// TIA Portal project "ELEVEYTOR" (V15.1)

(* hardware
DEVICE "S7-1200 station_1"  S7-1200 Station
   slot 0: "Rack_0"  S7-1200 Rack  Rack  V1.0
   slot 1: "PLC_1"  CPU 1214C AC/DC/Rly  6ES7 214-1BG40-0XB0  V4.2
   slot 2: "DI 16/DQ 16x24VDC_1"  6ES7 223-1BL32-0XB0  V2.0
DEVICE "PC-System_1"  SIMATIC PC station
   slot 0: "SIMATIC PC station"  Rail  SIMATIC PC-Station  V1.0
      slot 125: "Stationmanager"  Station_Manager  V6.0.4
   slot 1: "HMI_RT_1"  WinCC RT Advanced  6AV2 104-0xxxx-xxxx  15.1.0.0
      slot 33792: "Host interface"  Host interface
   slot 2: "IE general_1"  IE General  IE_CP  V8.2.0
*)

// ===== PLC "PLC_1"  CPU 1214C AC/DC/Rly =====

VAR_GLOBAL   // PLC tag table "Default tag table"
   "System_Byte" AT %MB1 : Byte;
   "FirstScan" AT %M1.0 : Bool;
   "DiagStatusUpdate" AT %M1.1 : Bool;
   "AlwaysTRUE" AT %M1.2 : Bool;
   "AlwaysFALSE" AT %M1.3 : Bool;
   "Clock_Byte" AT %MB0 : Byte;
   "Clock_10Hz" AT %M0.0 : Bool;
   "Clock_5Hz" AT %M0.1 : Bool;
   "Clock_2.5Hz" AT %M0.2 : Bool;
   "Clock_2Hz" AT %M0.3 : Bool;
   "Clock_1.25Hz" AT %M0.4 : Bool;
   "Clock_1Hz" AT %M0.5 : Bool;
   "Clock_0.625Hz" AT %M0.6 : Bool;
   "Clock_0.5Hz" AT %M0.7 : Bool;
   "Tag_1" AT %M900.0 : Bool;
   "Led" AT %MB6 : Byte;
END_VAR

VAR_GLOBAL   // PLC tag table "PRIORITIZE"
   "PRIORITIZE_1" AT %MB50 : SInt;   // Gọi lên x1, gọi xuống x0 (21,31, 41,51...20,30,40,50)
   "PRIORITIZE_2" AT %MB51 : SInt;
   "PRIORITIZE_3" AT %MB52 : SInt;
   "PRIORITIZE_4" AT %MB53 : SInt;
   "PRIORITIZE_5" AT %MB54 : SInt;
   "PRIORITIZE_6" AT %MB55 : SInt;
   "PRIORITIZE_SHIFT_1" AT %MD50 : DInt;
   "PRIORITIZE_SHIFT_2" AT %MD53 : DInt;
   "PRIORITIZE_SHIFT_3" AT %MD56 : DInt;
   "PRIORITIZE_7" AT %MB56 : SInt;
   "PRIORITIZE_8" AT %MB57 : SInt;
   "PRIORITIZE_9" AT %MB58 : SInt;
   "PRIORITIZE_10" AT %MB59 : SInt;
   "PRIORITIZE_11" AT %MB60 : SInt;
   "PRIORITIZE_12" AT %MB61 : SInt;
   "PRIORITIZE_SHIFT_4" AT %MD59 : DInt;
   "PRIORITIZE_POSITION" AT %MW70 : Int;
   "PRIORITIZE_13_Addition" AT %MB63 : SInt;   // Khi một tầng chọn cả lên và xuống thì dùng
   "PRIORITIZE_14_Addition" AT %MB64 : SInt;   // Spare
   "PRIORITIZE_15_Addition" AT %MB65 : SInt;   // Spare
   "PRIORITIZE_16_Addition" AT %MB66 : SInt;   // Spare
   "PRIORITIZE_SHIFT_5" AT %MD62 : DInt;
END_VAR

VAR_GLOBAL   // PLC tag table "OUTPUT"
   "Q_Lamp_System" AT %Q0.0 : Bool;   // Đèn làm việc
   "Q_Cabinet_Up" AT %Q0.1 : Bool;   // Buồng thang đi lên
   "Q_Cabinet_Down" AT %Q0.2 : Bool;   // Buồng thang đi xuống
   "Q_Door_Open" AT %Q0.3 : Bool;   // Cửa buồng thang mở
   "Q_Door_Close" AT %Q0.4 : Bool;   // Cửa buồng thang đóng
   "Q_BTT_Up_F1" AT %Q0.5 : Bool;   // Đèn nút nhấn đi lên F1
   "Q_BTT_Up_F2" AT %Q0.6 : Bool;   // Đèn nút nhấn đi lên F2
   "Q_BTT_Up_F3" AT %Q0.7 : Bool;   // Đèn nút nhấn đi lên F3
   "Q_BTT_Up_F4" AT %Q1.0 : Bool;   // Đèn nút nhấn đi lên F4
   "Q_BTT_Up_F5" AT %Q1.1 : Bool;   // Đèn nút nhấn đi lên F5
   "Q_BTT_Down_F2" AT %Q1.2 : Bool;   // Đèn nút nhấn đi xuống F2
   "Q_BTT_Down_F3" AT %Q1.3 : Bool;   // Đèn nút nhấn đi xuống F3
   "Q_BTT_Down_F4" AT %Q1.4 : Bool;   // Đèn nút nhấn đi xuống F4
   "Q_BTT_Down_F5" AT %Q1.5 : Bool;   // Đèn nút nhấn đi xuống F5
   "Q_BTT_Down_F6" AT %Q1.6 : Bool;   // Đèn nút nhấn đi xuống F6
   "Q_BTT_CABIN_F1" AT %Q1.7 : Bool;   // Đèn nút nhấn trong buồng thang F1
   "Q_BTT_CABIN_F2" AT %Q2.0 : Bool;   // Đèn nút nhấn trong buồng thang F2
   "Q_BTT_CABIN_F3" AT %Q2.1 : Bool;   // Đèn nút nhấn trong buồng thang F3
   "Q_BTT_CABIN_F4" AT %Q2.2 : Bool;   // Đèn nút nhấn trong buồng thang F4
   "Q_BTT_CABIN_F5" AT %Q2.3 : Bool;   // Đèn nút nhấn trong buồng thang F5
   "Q_BTT_CABIN_F6" AT %Q2.4 : Bool;   // Đèn nút nhấn trong buồng thang F6
   "Q_Lamp_Weight_Alarm" AT %Q2.5 : Bool;   // Đèn cảnh báo quá trọng lượng
END_VAR

VAR_GLOBAL   // PLC tag table "INPUT"
   "I_BTT_DOOR_OPEN" AT %I1.4 : Bool;   // Nút nhấn mở cửa
   "I_BTT_DOOR_CLOSE" AT %I2.7 : Bool;   // Nút nhấn đóng cửa
   "I_BTT_CABINET_F1" AT %I0.5 : Bool;   // Nút nhấn chọn tầng trong thang máy Tầng 1
   "I_BTT_CABINET_F2" AT %I0.3 : Bool;   // Nút nhấn chọn tầng trong thang máy Tầng 2
   "I_BTT_CABINET_F3" AT %I0.2 : Bool;   // Nút nhấn chọn tầng trong thang máy Tầng 3
   "I_BTT_CABINET_F4" AT %I0.4 : Bool;   // Nút nhấn chọn tầng trong thang máy Tầng 4
   "I_BTT_UP_F1" AT %I1.2 : Bool;   // Nút nhấn đi lên/xuống tầng 1
   "I_BTT_UP_F2" AT %I0.6 : Bool;   // Nút nhấn đi lên tầng 2
   "I_BTT_UP_F3" AT %I1.0 : Bool;   // Nút nhấn đi lên tầng 3
   "I_BTT_DOWN_F2" AT %I1.3 : Bool;   // Nút nhấn đi xuống tầng 2
   "I_BTT_DOWN_F3" AT %I0.7 : Bool;   // Nút nhấn đi xuống tầng 3
   "I_BTT_DOWN_F4" AT %I1.1 : Bool;   // Nút nhấn đi xuống tầng 4
   "I_LS_DOOR_OPENED" AT %I2.5 : Bool;   // Công tắc hành trình mở cửa
   "I_LS_DOOR_CLOSED" AT %I2.4 : Bool;   // Công tắc hành trình đóng cửa
   "I_BTT_MAN_CABINET_UP" AT %I3.0 : Bool;   // Nút nhấn cabinet nâng chế độ bằng tay
   "I_BTT_MAN_CABINET_DOWN" AT %I2.6 : Bool;   // Nút nhấn cabinet hạ chế độ bằng tay
   "I_BTT_MAN_DOOR_OPEN" AT %I3.1 : Bool;   // Nút nhấn mở cửa chế độ bằng tay
   "I_BTT_MAN_DOOR_CLOSE" AT %I3.5 : Bool;   // nút nhấn đóng cửa chế độ bằng tay
   "I_SW_AUTO" AT %I3.6 : Bool;   // Switch chọn chế độ tự động
   "I_SW_MANU" AT %I3.2 : Bool;   // Switch chọn chế độ bằng tay
   "ID0" AT %ID0 : DWord;
   "I_BTT_MAN_CABIN_STOP" AT %I13.3 : Bool;
   "I_LS_CABINET_2" AT %I2.1 : Bool;
   "I_LS_CABINET_3" AT %I2.2 : Bool;
   "I_LS_CABINET_4" AT %I2.3 : Bool;
   "I_LS_CABINET_1" AT %I2.0 : Bool;
END_VAR

VAR_GLOBAL   // PLC tag table "MEMORY"
   "M_BTT_DOOR_OPEN" AT %M10.0 : Bool;
   "M_BTT_DOOR_CLOSE" AT %M10.1 : Bool;
   "M_BTT_CABINET_F1" AT %M10.2 : Bool;
   "M_BTT_CABINET_F2" AT %M10.3 : Bool;
   "M_BTT_CABINET_F3" AT %M10.4 : Bool;
   "M_BTT_CABINET_F4" AT %M10.5 : Bool;
   "M_BTT_CABINET_F5" AT %M10.6 : Bool;
   "M_BTT_CABINET_F6" AT %M10.7 : Bool;
   "M_BTT_UP_F1" AT %M11.0 : Bool;
   "M_BTT_UP_F2" AT %M11.1 : Bool;
   "M_BTT_UP_F3" AT %M11.2 : Bool;
   "M_BTT_UP_F4" AT %M11.3 : Bool;
   "M_BTT_UP_F5" AT %M11.4 : Bool;
   "M_BTT_DOWN_F2" AT %M11.5 : Bool;
   "M_BTT_DOWN_F3" AT %M11.6 : Bool;
   "M_BTT_DOWN_F4" AT %M11.7 : Bool;
   "M_BTT_DOWN_F5" AT %M12.0 : Bool;
   "M_BTT_DOWN_F6" AT %M12.1 : Bool;
   "M_LS_CABINET" AT %M12.2 : Bool;
   "M_LS_DOOR_OPENED" AT %M12.3 : Bool;
   "M_LS_DOOR_CLOSED" AT %M12.4 : Bool;
   "M_BTT_MAN_CABINET_UP" AT %M12.5 : Bool;
   "M_BTT_MAN_CABINET_DOWN" AT %M12.6 : Bool;
   "M_BTT_MAN_DOOR_OPEN" AT %M12.7 : Bool;
   "M_BTT_MAN_DOOR_CLOSE" AT %M13.0 : Bool;
   "M_SW_AUTO" AT %M13.1 : Bool;
   "M_SW_MANU" AT %M13.2 : Bool;
   "M_BTT_Simulation" AT %M300.0 : Bool;
   "MD10" AT %MD10 : DWord;
   "M_BTT_MAN_DOOR_STOP" AT %M13.4 : Bool;
   "M_BTT_MAN_CABIN_STOP" AT %M13.3 : Bool;
END_VAR

DATA_BLOCK "DB_Status"   // DB1
{ S7_Optimized_Access := 'FALSE' }
VERSION : 0.1
   VAR
      PRIOTIZE_1 : SInt;
      PRIOTIZE_2 : SInt;
      PRIOTIZE_3 : SInt;
      PRIOTIZE_4 : SInt;
      PRIOTIZE_5 : SInt;
      PRIOTIZE_6 : SInt;
      PRIOTIZE_7 : SInt;
      PRIOTIZE_8 : SInt;
      PRIOTIZE_9 : SInt;
      PRIOTIZE_10 : SInt;
      PRIOTIZE_11 : SInt;
      PRIOTIZE_12 : SInt;
      PRIOTIZE_13 : SInt;
      PRIOTIZE_14 : SInt;
      PRIOTIZE_15 : SInt;
      PRIOTIZE_16 : SInt;
      PRIOTIZE_17 : SInt;
      PRIOTIZE_18 : SInt;
      PRIOTIZE_19 : SInt;
      PRIOTIZE_20 : SInt;
      LS_F1 : Bool;
      LS_F2 : Bool;
      LS_F3 : Bool;
      LS_F4 : Bool;
      LS_F5 : Bool;
      LS_F6 : Bool;
      LS_F7 : Bool;   // Spare
      LS_F8 : Bool;   // Spare
      LS_F9 : Bool;   // Spare
      LS_F10 : Bool;   // Spare
      Up_Called_F1 : Bool;
      Up_Called_F2 : Bool;
      Up_Called_F3 : Bool;
      Up_Called_F4 : Bool;
      Up_Called_F5 : Bool;
      Up_Called_F6 : Bool;
      Down_Called_F1 : Bool;
      Down_Called_F2 : Bool;
      Down_Called_F3 : Bool;
      Down_Called_F4 : Bool;
      Down_Called_F5 : Bool;
      Down_Called_F6 : Bool;
      Q_Lamp_System : Bool;
      Q_Cabinet_Up : Bool;
      Q_Cabinet_Down : Bool;
      Q_Door_Open : Bool;
      Q_Door_Close : Bool;
      Q_BTT_Up_F1 : Bool;
      Q_BTT_Up_F2 : Bool;
      Q_BTT_Up_F3 : Bool;
      Q_BTT_Up_F4 : Bool;
      Q_BTT_Up_F5 : Bool;
      Q_BTT_Down_F2 : Bool;
      Q_BTT_Down_F3 : Bool;
      Q_BTT_Down_F4 : Bool;
      Q_BTT_Down_F5 : Bool;
      Q_BTT_Down_F6 : Bool;
      DOOR_Delay_Open : Bool;
      CABINET_AT_FLOOR : Int;
      Actual_Weight : Real;
      CABIN_LastStatus_Upping : Bool;   // Trước đó buồng thang đi lên (trạng thái)
      CABIN_LastStatus_Dowing : Bool;   // Trước đó buồng thang đi xuống (trạng thái)
   END_VAR
BEGIN
END_DATA_BLOCK

DATA_BLOCK "DB_PRIOTIZE"   // DB2
{ S7_Optimized_Access := 'TRUE' }
VERSION : 0.1
BEGIN
END_DATA_BLOCK

DATA_BLOCK "DB_Command"   // DB3
{ S7_Optimized_Access := 'TRUE' }
VERSION : 0.1
   VAR
      F1_Up_Seleced : Bool;
      F2_Up_Seleced : Bool;
      F3_Up_Seleced : Bool;
      F4_Up_Seleced : Bool;
      F5_Up_Seleced : Bool;
      F2_Down_Seleced : Bool;
      F3_Down_Seleced : Bool;
      F4_Down_Seleced : Bool;
      F5_Down_Seleced : Bool;
      F6_Down_Seleced : Bool;
      F1_Selected : Bool;
      F2_Selected : Bool;
      F3_Selected : Bool;
      F4_Selected : Bool;
      F5_Selected : Bool;
      F6_Selected : Bool;
      F_Rq_Cabin_Stop : Bool;   // Yêu cầu dừng cabin FC tầng gọi cuối cùng
      F_Rq_Door_Open : Bool;   // Yêu cầu mở cửa FC tầng gọi cuối cùng
      F_Rq_Clear_Priotize : Bool;   // Yêu cầu xóa ưu tiên FC tầng gọi cuối cùng
   END_VAR
BEGIN
END_DATA_BLOCK

DATA_BLOCK "PULSE"   // DB4
{ S7_Optimized_Access := 'TRUE' }
VERSION : 0.1
   VAR
      FC2_F1_P1 : Bool;
      FC2_F1_P2 : Bool;
      FC2_F2_P1 : Bool;
      FC2_F2_P2 : Bool;
      FC2_F3_P1 : Bool;
      FC2_F3_P2 : Bool;
      FC2_F4_P1 : Bool;
      FC2_F4_P2 : Bool;
      FC2_F5_P1 : Bool;
      FC2_F5_P2 : Bool;
      FC2_F6_P1 : Bool;
      FC2_F6_P2 : Bool;
      FC1_P1 : Bool;
      FC1_P2 : Bool;
      F1_Upping_P1 : Bool;
      F1_Upping_P2 : Bool;
      F2_Upping_P1 : Bool;
      F2_Upping_P2 : Bool;
      F3_Upping_P1 : Bool;
      F3_Upping_P2 : Bool;
      F4_Upping_P1 : Bool;
      F4_Upping_P2 : Bool;
      F5_Upping_P1 : Bool;
      F5_Upping_P2 : Bool;
      F6_Upping_P1 : Bool;
      F6_Upping_P2 : Bool;
      F1_Downing_P1 : Bool;
      F1_Downing_P2 : Bool;
      F2_Downing_P1 : Bool;
      F2_Downing_P2 : Bool;
      F3_Downing_P1 : Bool;
      F3_Downing_P2 : Bool;
      F4_Downing_P1 : Bool;
      F4_Downing_P2 : Bool;
      F5_Downing_P1 : Bool;
      F5_Downing_P2 : Bool;
      F6_Downing_P1 : Bool;
      F6_Downing_P2 : Bool;
      FC7_N1 : Bool;
      FC7_P1 : Bool;
      FC7_P2 : Bool;
      FC7_P3 : Bool;
      FC7_P4 : Bool;
      FC7_N2 : Bool;
      FC7_P5 : Bool;
      FC7_Pulse_Door_Lock : Bool;
      FC7_N3 : Bool;
      FC12_Pulse_2S : Bool;
      "2Second_Pulse_Upping_F1" : Bool;
      "2Second_Pulse_Upping_F2" : Bool;
      "2Second_Pulse_Upping_F3" : Bool;
      "2Second_Pulse_Upping_F4" : Bool;
      "2Second_Pulse_Upping_F5" : Bool;
      "2Second_Pulse_Upping_F6" : Bool;
      "2Second_Pulse_Downing_F1" : Bool;
      "2Second_Pulse_Downing_F2" : Bool;
      "2Second_Pulse_Downing_F3" : Bool;
      "2Second_Pulse_Downing_F4" : Bool;
      "2Second_Pulse_Downing_F5" : Bool;
      "2Second_Pulse_Downing_F6" : Bool;
      FC4_Temp_Pulse : Bool;
      FC12_Pulse_Up_F1 : Bool;
      FC12_Pulse_Up_F2 : Bool;
      FC12_Pulse_Up_F3 : Bool;
      FC12_Pulse_Up_F4 : Bool;
      FC12_Pulse_Up_F5 : Bool;
      FC12_Pulse_Up_F6 : Bool;
      FC12_Pulse_Down_F1 : Bool;
      FC12_Pulse_Down_F2 : Bool;
      FC12_Pulse_Down_F3 : Bool;
      FC12_Pulse_Down_F4 : Bool;
      FC12_Pulse_Down_F5 : Bool;
      FC12_Pulse_Down_F6 : Bool;
      FC7_Pulse_Door_Lock_Temp : Bool;
      FC8_P1 : Bool;
      FC8_P2 : Bool;
      FC1_P3 : Bool;
      FC1_Shift_Request : Bool;
   END_VAR
BEGIN
END_DATA_BLOCK

DATA_BLOCK "DB_FRECONDITION"   // DB5
{ S7_Optimized_Access := 'TRUE' }
VERSION : 0.1
   VAR
      DOOR_Open : Bool;
      DOOR_Permit_time : Bool;
   END_VAR
BEGIN
END_DATA_BLOCK

DATA_BLOCK "DB_SETTING"   // DB6
{ S7_Optimized_Access := 'TRUE' }
VERSION : 0.1
   VAR RETAIN
      Weight : Real := 1000.0;
      Door_Open_Time : Time := T#5ms;
      Extreme_Time : Time := T#5ms;
   END_VAR
BEGIN
END_DATA_BLOCK

DATA_BLOCK "DB_SIMULATION"   // DB8
{ S7_Optimized_Access := 'TRUE' }
VERSION : 0.1
   VAR
      POS_CABINET : Int;
      POS_DOOR : Int;
      DOOR_F1 : Int;   // THANG MÁY Ở TẦNG 1
      DOOR_F2 : Int;   // THANG MÁY Ở TẦNG 2
      DOOR_F3 : Int;   // THANG MÁY Ở TẦNG 3
      DOOR_F4 : Int;   // THANG MÁY Ở TẦNG 4
      Weight : DInt;
   END_VAR
BEGIN
END_DATA_BLOCK

DATA_BLOCK "Display_number_DB"   // DB15
{ S7_Optimized_Access := 'TRUE' }
VERSION : 0.1
// stored: InstanceOfName Display_number
"Display_number"
BEGIN
END_DATA_BLOCK

// folder: System blocks/Program resources

DATA_BLOCK "DELAY_OPEN"   // DB7
{ S7_Optimized_Access := 'TRUE' }
AUTHOR : Simatic
FAMILY : IEC
NAME : IEC_TMR
VERSION : 1.0
// stored: InstanceOfName IEC_TIMER
"IEC_TIMER"
BEGIN
END_DATA_BLOCK

DATA_BLOCK "SIMU_CABINET"   // DB9
{ S7_Optimized_Access := 'TRUE' }
AUTHOR : Simatic
FAMILY : IEC
NAME : CNTR
VERSION : 1.0
// stored: InstanceOfName IEC_COUNTER
"IEC_COUNTER"
BEGIN
END_DATA_BLOCK

DATA_BLOCK "SIMU_DOOR"   // DB10
{ S7_Optimized_Access := 'TRUE' }
AUTHOR : Simatic
FAMILY : IEC
NAME : CNTR
VERSION : 1.0
// stored: InstanceOfName IEC_COUNTER
"IEC_COUNTER"
BEGIN
END_DATA_BLOCK

DATA_BLOCK "DOOR_EXTREME"   // DB11
{ S7_Optimized_Access := 'TRUE' }
AUTHOR : Simatic
FAMILY : IEC
NAME : IEC_TMR
VERSION : 1.0
// stored: InstanceOfName IEC_TIMER
"IEC_TIMER"
BEGIN
END_DATA_BLOCK

DATA_BLOCK "FC12_DELAY_2S"   // DB12
{ S7_Optimized_Access := 'TRUE' }
AUTHOR : Simatic
FAMILY : IEC
NAME : IEC_TMR
VERSION : 1.0
// stored: InstanceOfName IEC_TIMER
"IEC_TIMER"
BEGIN
END_DATA_BLOCK

DATA_BLOCK "FC4_PULSE_2S"   // DB13
{ S7_Optimized_Access := 'TRUE' }
AUTHOR : Simatic
FAMILY : IEC
NAME : IEC_TMR
VERSION : 1.0
// stored: InstanceOfName IEC_TIMER
"IEC_TIMER"
BEGIN
END_DATA_BLOCK

DATA_BLOCK "PULSE_DOOR_LOCK"   // DB14
{ S7_Optimized_Access := 'TRUE' }
AUTHOR : Simatic
FAMILY : IEC
NAME : IEC_TMR
VERSION : 1.0
// stored: InstanceOfName IEC_TIMER
"IEC_TIMER"
BEGIN
END_DATA_BLOCK

// folder: (top level)

FUNCTION_BLOCK "Display_number"   // FB1, SCL
{ S7_Optimized_Access := 'TRUE' }
VERSION : 0.1
   VAR_INPUT
      BCD : Int;
   END_VAR
   VAR_OUTPUT
      LED : Byte;
   END_VAR
   VAR_TEMP
      TMP : Byte;
   END_VAR
BEGIN
   CASE #BCD OF
       1:  // Statement section case 1
           #TMP := 16#6;
       2:  // Statement section case 1
           #TMP := 16#5B;
       3:  // Statement section case 1
           #TMP := 16#4F;
       4:  // Statement section case 1
           #TMP := 16#66;

       ELSE  // Statement section ELSE
           ;
   END_CASE;
   #LED := #TMP;
END_FUNCTION_BLOCK

FUNCTION "1.FC_SHIFT" : Void   // FC1, LAD
{ S7_Optimized_Access := 'TRUE' }
VERSION : 0.1
// 1. Network 1 là lệnh shift word (tức là di chuyển chể độ ưu tiên), ở đây sẽ có 6 chế độ ưu tiên, tầng nào ưu tiên nhất thì sẽ ưu tiên tầng đó.
// Bit shift sẽ thực hiện khi:
// 1.1. Thang máy chạm công tắc hành trình của một tầng nào đó
// 1.2. Cửa buồng thang mở
// >>> tất nhiên với điều kiện ở ô nhớ ưu tiên 1 không phải là tầng đó, ví dụ đang ở tầng 2 mà ô nhớ ưu tiên 1 có giá trị là 2 thì mới shift, còn không thì thôi.
// 
// >>> Nếu giá trị ưu tiên đầu tiên mà bằng 0 thì tiến hành shift các miền nhớ khác tiến về trước mỗi 100ms (Clock_10Hz)
   VAR_TEMP   // added for the SCL form of the ladder/FBD networks
      _w1 : Bool;
      _w2 : Bool;
   END_VAR
BEGIN

REGION Network 1: SHIFT PRIORITIZE
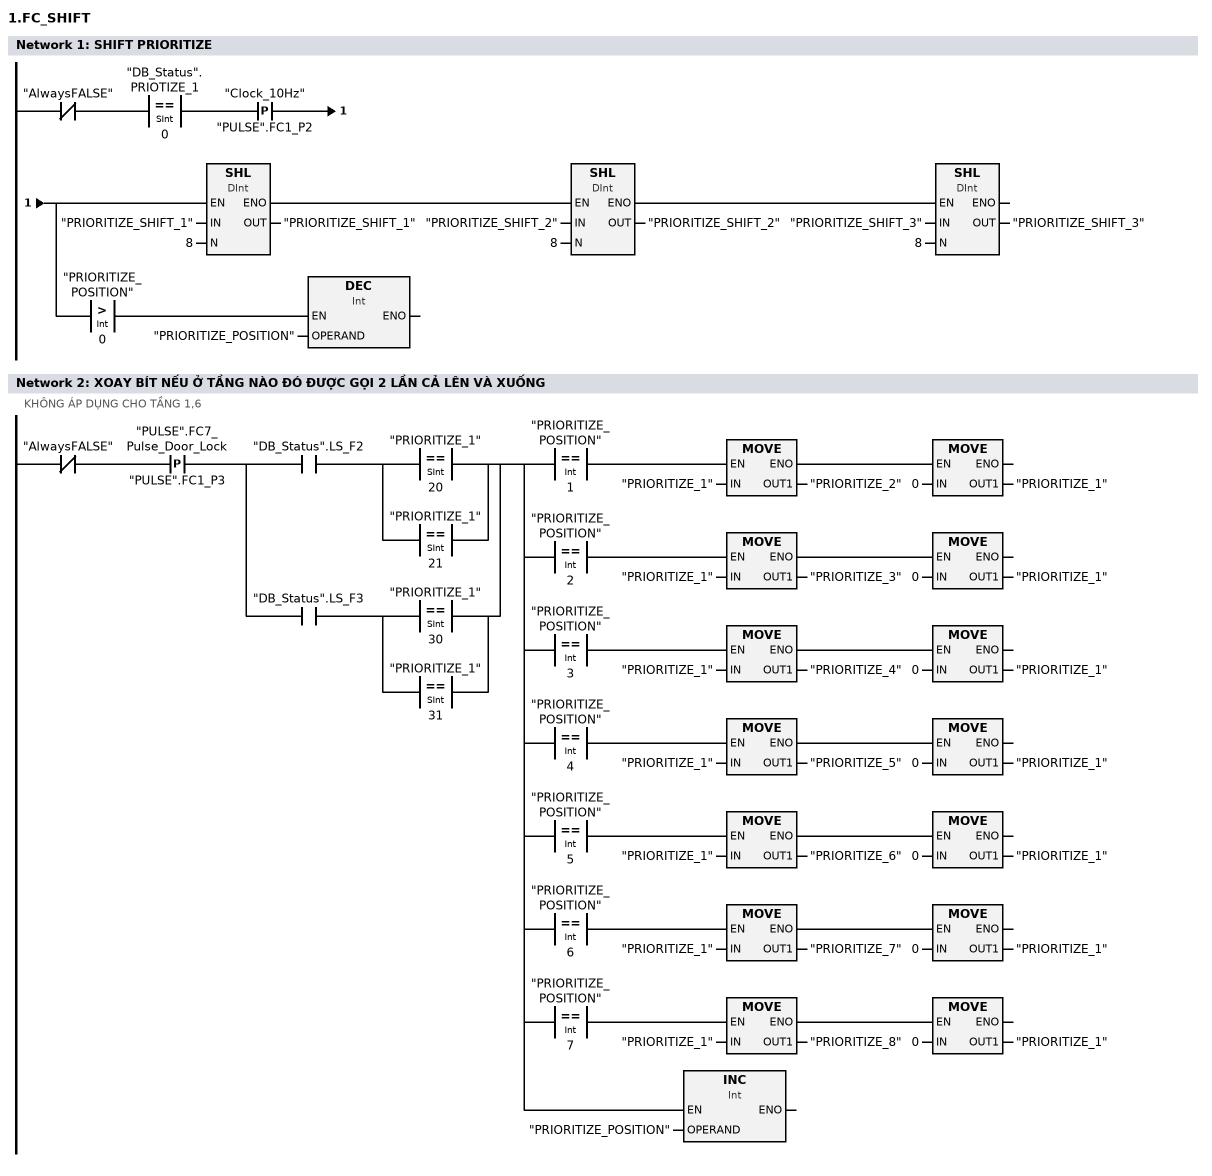
   RUNG wire#powerrail
      I_Contact( "AlwaysFALSE" )
      { S7_Templates := "SrcType := SInt" } EQ_Contact(in1 := "DB_Status".PRIOTIZE_1, in2 := 0)
      P_Contact(operand := "Clock_10Hz", bit := "PULSE".FC1_P2)
      wire#w1
      { S7_Templates := "SrcType := DInt" } Shl(in := "PRIORITIZE_SHIFT_1", n := 8, out => "PRIORITIZE_SHIFT_1")
      { S7_Templates := "SrcType := DInt" } Shl(in := "PRIORITIZE_SHIFT_2", n := 8, out => "PRIORITIZE_SHIFT_2")
      { S7_Templates := "SrcType := DInt" } Shl(in := "PRIORITIZE_SHIFT_3", n := 8, out => "PRIORITIZE_SHIFT_3")
   END_RUNG
   RUNG wire#w1
      { S7_Templates := "SrcType := Int" } GT_Contact(in1 := "PRIORITIZE_POSITION", in2 := 0)
      { S7_Templates := "DestType := Int" } Dec( "PRIORITIZE_POSITION" )
   END_RUNG
   // the same network as SCL:
   #_w1 := NOT "AlwaysFALSE" AND ("DB_Status".PRIOTIZE_1 = 0) AND "Clock_10Hz" AND NOT "PULSE".FC1_P2;   // rising edge of "Clock_10Hz"
   "PULSE".FC1_P2 := "Clock_10Hz";
   IF #_w1 THEN
       "PRIORITIZE_SHIFT_1" := SHL(IN := "PRIORITIZE_SHIFT_1", N := 8);
       "PRIORITIZE_SHIFT_2" := SHL(IN := "PRIORITIZE_SHIFT_2", N := 8);
       "PRIORITIZE_SHIFT_3" := SHL(IN := "PRIORITIZE_SHIFT_3", N := 8);
   END_IF;
   IF #_w1 AND ("PRIORITIZE_POSITION" > 0) THEN "PRIORITIZE_POSITION" := "PRIORITIZE_POSITION" - 1; END_IF;
END_REGION

REGION Network 2: XOAY BÍT NẾU Ở TẦNG NÀO ĐÓ ĐƯỢC GỌI 2 LẦN CẢ LÊN VÀ XUỐNG
   // KHÔNG ÁP DỤNG CHO TẦNG 1,6
   RUNG wire#powerrail
      I_Contact( "AlwaysFALSE" )
      P_Contact(operand := "PULSE".FC7_Pulse_Door_Lock, bit := "PULSE".FC1_P3)
      wire#w1
      Contact( "DB_Status".LS_F2 )
      wire#w2
      { S7_Templates := "SrcType := SInt" } EQ_Contact(in1 := "PRIORITIZE_1", in2 := 20)
      wire#w3
      { S7_Templates := "SrcType := Int" } EQ_Contact(in1 := "PRIORITIZE_POSITION", in2 := 1)
      Move(in := "PRIORITIZE_1", out1 => "PRIORITIZE_2")
      Move(in := 0, out1 => "PRIORITIZE_1")
   END_RUNG
   RUNG wire#w2
      { S7_Templates := "SrcType := SInt" } EQ_Contact(in1 := "PRIORITIZE_1", in2 := 21)
   END_RUNG wire#w3
   RUNG wire#w1
      Contact( "DB_Status".LS_F3 )
      wire#w4
      { S7_Templates := "SrcType := SInt" } EQ_Contact(in1 := "PRIORITIZE_1", in2 := 30)
   END_RUNG wire#w3
   RUNG wire#w4
      { S7_Templates := "SrcType := SInt" } EQ_Contact(in1 := "PRIORITIZE_1", in2 := 31)
   END_RUNG wire#w3
   RUNG wire#w3
      { S7_Templates := "SrcType := Int" } EQ_Contact(in1 := "PRIORITIZE_POSITION", in2 := 2)
      Move(in := "PRIORITIZE_1", out1 => "PRIORITIZE_3")
      Move(in := 0, out1 => "PRIORITIZE_1")
   END_RUNG
   RUNG wire#w3
      { S7_Templates := "SrcType := Int" } EQ_Contact(in1 := "PRIORITIZE_POSITION", in2 := 3)
      Move(in := "PRIORITIZE_1", out1 => "PRIORITIZE_4")
      Move(in := 0, out1 => "PRIORITIZE_1")
   END_RUNG
   RUNG wire#w3
      { S7_Templates := "SrcType := Int" } EQ_Contact(in1 := "PRIORITIZE_POSITION", in2 := 4)
      Move(in := "PRIORITIZE_1", out1 => "PRIORITIZE_5")
      Move(in := 0, out1 => "PRIORITIZE_1")
   END_RUNG
   RUNG wire#w3
      { S7_Templates := "SrcType := Int" } EQ_Contact(in1 := "PRIORITIZE_POSITION", in2 := 5)
      Move(in := "PRIORITIZE_1", out1 => "PRIORITIZE_6")
      Move(in := 0, out1 => "PRIORITIZE_1")
   END_RUNG
   RUNG wire#w3
      { S7_Templates := "SrcType := Int" } EQ_Contact(in1 := "PRIORITIZE_POSITION", in2 := 6)
      Move(in := "PRIORITIZE_1", out1 => "PRIORITIZE_7")
      Move(in := 0, out1 => "PRIORITIZE_1")
   END_RUNG
   RUNG wire#w3
      { S7_Templates := "SrcType := Int" } EQ_Contact(in1 := "PRIORITIZE_POSITION", in2 := 7)
      Move(in := "PRIORITIZE_1", out1 => "PRIORITIZE_8")
      Move(in := 0, out1 => "PRIORITIZE_1")
   END_RUNG
   RUNG wire#w3
      { S7_Templates := "DestType := Int" } Inc( "PRIORITIZE_POSITION" )
   END_RUNG
   // the same network as SCL:
   #_w1 := NOT "AlwaysFALSE" AND "PULSE".FC7_Pulse_Door_Lock AND NOT "PULSE".FC1_P3;   // rising edge of "PULSE".FC7_Pulse_Door_Lock
   "PULSE".FC1_P3 := "PULSE".FC7_Pulse_Door_Lock;
   #_w2 := #_w1 AND (("DB_Status".LS_F2 AND (("PRIORITIZE_1" = 20) OR ("PRIORITIZE_1" = 21))) OR ("DB_Status".LS_F3 AND (("PRIORITIZE_1" = 30) OR ("PRIORITIZE_1" = 31))));
   IF #_w2 AND ("PRIORITIZE_POSITION" = 1) THEN
       "PRIORITIZE_2" := "PRIORITIZE_1";
       "PRIORITIZE_1" := 0;
   END_IF;
   IF #_w2 AND ("PRIORITIZE_POSITION" = 2) THEN
       "PRIORITIZE_3" := "PRIORITIZE_1";
       "PRIORITIZE_1" := 0;
   END_IF;
   IF #_w2 AND ("PRIORITIZE_POSITION" = 3) THEN
       "PRIORITIZE_4" := "PRIORITIZE_1";
       "PRIORITIZE_1" := 0;
   END_IF;
   IF #_w2 AND ("PRIORITIZE_POSITION" = 4) THEN
       "PRIORITIZE_5" := "PRIORITIZE_1";
       "PRIORITIZE_1" := 0;
   END_IF;
   IF #_w2 AND ("PRIORITIZE_POSITION" = 5) THEN
       "PRIORITIZE_6" := "PRIORITIZE_1";
       "PRIORITIZE_1" := 0;
   END_IF;
   IF #_w2 AND ("PRIORITIZE_POSITION" = 6) THEN
       "PRIORITIZE_7" := "PRIORITIZE_1";
       "PRIORITIZE_1" := 0;
   END_IF;
   IF #_w2 AND ("PRIORITIZE_POSITION" = 7) THEN
       "PRIORITIZE_8" := "PRIORITIZE_1";
       "PRIORITIZE_1" := 0;
   END_IF;
   IF #_w2 THEN "PRIORITIZE_POSITION" := "PRIORITIZE_POSITION" + 1; END_IF;
END_REGION
END_FUNCTION

FUNCTION "2.FC_PRIOTIZE" : Void   // FC2, SCL
{ S7_Optimized_Access := 'TRUE' }
VERSION : 0.1
   VAR_INPUT
      F1_Up_Selected : Bool;
      F2_Up_Selected : Bool;
      F3_Up_Selected : Bool;
      F4_Up_Selected : Bool;
      F4_Down_Selected : Bool;
      F3_Down_Selected : Bool;
      F2_Down_Selected : Bool;
   END_VAR
   VAR_OUTPUT
      PRI_1 : SInt;
      PRI_2 : SInt;
      PRI_3 : SInt;
      PRI_4 : SInt;
      PRI_5 : SInt;
      PRI_6 : SInt;
      PRI_7 : SInt;
      PRI_8 : SInt;
   END_VAR
   VAR_IN_OUT
      PRIORITIZE_POSITION : Int;
   END_VAR
BEGIN
   // Đầu vào nhơ đặt xung sườn lên cho các INPUT
   //Thực hiện chọn tầng ưu tiên từ ưu tiên 1 đến ưu tiên 6, lệnh sẽ thực hiện khi nhấn nút chọn tầng (lên hoặc xuống)
   //Đưa giá trị ưu tiên ra đầu ra của chương trình con
   // F1 CHỌN ĐI LÊN
   IF #F1_Up_Selected = TRUE THEN
       IF #PRIORITIZE_POSITION = 0 THEN
           "PRIORITIZE_1" := 11;
           #PRIORITIZE_POSITION := 1;
       ELSIF #PRIORITIZE_POSITION = 1 THEN
           "PRIORITIZE_2" := 11;
           #PRIORITIZE_POSITION := 2;
       ELSIF #PRIORITIZE_POSITION = 2 THEN
           "PRIORITIZE_3" := 11;
           #PRIORITIZE_POSITION := 3;
       ELSIF #PRIORITIZE_POSITION = 3 THEN
           "PRIORITIZE_4" := 11;
           #PRIORITIZE_POSITION := 4;
       ELSIF #PRIORITIZE_POSITION = 4 THEN
           "PRIORITIZE_5" := 11;
           #PRIORITIZE_POSITION := 5;
       ELSIF #PRIORITIZE_POSITION = 5 THEN
           "PRIORITIZE_6" := 11;
           #PRIORITIZE_POSITION := 6;
       ELSIF #PRIORITIZE_POSITION = 6 THEN
           "PRIORITIZE_7" := 11;
           #PRIORITIZE_POSITION := 7;
       ELSIF #PRIORITIZE_POSITION = 7 THEN
           "PRIORITIZE_8" := 11;
           #PRIORITIZE_POSITION := 8;

           ;
       END_IF;
       ;
   END_IF;
   // F2 CHỌN ĐI LÊN
   IF #F2_Up_Selected = TRUE THEN
       IF #PRIORITIZE_POSITION = 0 THEN
           "PRIORITIZE_1" := 21;
           #PRIORITIZE_POSITION := 1;
       ELSIF #PRIORITIZE_POSITION = 1 THEN
           "PRIORITIZE_2" := 21;
           #PRIORITIZE_POSITION := 2;
       ELSIF #PRIORITIZE_POSITION = 2 THEN
           "PRIORITIZE_3" := 21;
           #PRIORITIZE_POSITION := 3;
       ELSIF #PRIORITIZE_POSITION = 3 THEN
           "PRIORITIZE_4" := 21;
           #PRIORITIZE_POSITION := 4;
       ELSIF #PRIORITIZE_POSITION = 4 THEN
           "PRIORITIZE_5" := 21;
           #PRIORITIZE_POSITION := 5;
       ELSIF #PRIORITIZE_POSITION = 5 THEN
           "PRIORITIZE_6" := 21;
           #PRIORITIZE_POSITION := 6;
       ELSIF #PRIORITIZE_POSITION = 6 THEN
           "PRIORITIZE_7" := 21;
           #PRIORITIZE_POSITION := 7;
       ELSIF #PRIORITIZE_POSITION = 7 THEN
           "PRIORITIZE_8" := 21;
           #PRIORITIZE_POSITION := 8;

           ;
       END_IF;
       ;
   END_IF;
   // F3 ĐI LÊN
   IF #F3_Up_Selected = TRUE THEN
       IF #PRIORITIZE_POSITION = 0 THEN
           "PRIORITIZE_1" := 31;
           #PRIORITIZE_POSITION := 1;
       ELSIF #PRIORITIZE_POSITION = 1 THEN
           "PRIORITIZE_2" := 31;
           #PRIORITIZE_POSITION := 2;
       ELSIF #PRIORITIZE_POSITION = 2 THEN
           "PRIORITIZE_3" := 31;
           #PRIORITIZE_POSITION := 3;
       ELSIF #PRIORITIZE_POSITION = 3 THEN
           "PRIORITIZE_4" := 31;
           #PRIORITIZE_POSITION := 4;
       ELSIF #PRIORITIZE_POSITION = 4 THEN
           "PRIORITIZE_5" := 31;
           #PRIORITIZE_POSITION := 5;
       ELSIF #PRIORITIZE_POSITION = 5 THEN
           "PRIORITIZE_6" := 31;
           #PRIORITIZE_POSITION := 6;
       ELSIF #PRIORITIZE_POSITION = 6 THEN
           "PRIORITIZE_7" := 31;
           #PRIORITIZE_POSITION := 7;
       ELSIF #PRIORITIZE_POSITION = 7 THEN
           "PRIORITIZE_8" := 31;
           #PRIORITIZE_POSITION := 8;

           ;
       END_IF;
       ;
   END_IF;
   // F4 ĐI LÊN
   IF #F4_Up_Selected = TRUE THEN
       IF #PRIORITIZE_POSITION = 0 THEN
           "PRIORITIZE_1" := 41;
           #PRIORITIZE_POSITION := 1;
       ELSIF #PRIORITIZE_POSITION = 1 THEN
           "PRIORITIZE_2" := 41;
           #PRIORITIZE_POSITION := 2;
       ELSIF #PRIORITIZE_POSITION = 2 THEN
           "PRIORITIZE_3" := 41;
           #PRIORITIZE_POSITION := 3;
       ELSIF #PRIORITIZE_POSITION = 3 THEN
           "PRIORITIZE_4" := 41;
           #PRIORITIZE_POSITION := 4;
       ELSIF #PRIORITIZE_POSITION = 4 THEN
           "PRIORITIZE_5" := 41;
           #PRIORITIZE_POSITION := 5;
       ELSIF #PRIORITIZE_POSITION = 5 THEN
           "PRIORITIZE_6" := 41;
           #PRIORITIZE_POSITION := 6;
       ELSIF #PRIORITIZE_POSITION = 6 THEN
           "PRIORITIZE_7" := 41;
           #PRIORITIZE_POSITION := 7;
       ELSIF #PRIORITIZE_POSITION = 7 THEN
           "PRIORITIZE_8" := 41;
           #PRIORITIZE_POSITION := 8;

           ;
       END_IF;
       ;
   END_IF;


   //F4 ĐI XUỐNG
   IF #F4_Down_Selected = TRUE THEN
       IF #PRIORITIZE_POSITION = 0 THEN
           "PRIORITIZE_1" := 40;
           #PRIORITIZE_POSITION := 1;
       ELSIF #PRIORITIZE_POSITION = 1 THEN
           "PRIORITIZE_2" := 40;
           #PRIORITIZE_POSITION := 2;
       ELSIF #PRIORITIZE_POSITION = 2 THEN
           "PRIORITIZE_3" := 40;
           #PRIORITIZE_POSITION := 3;
       ELSIF #PRIORITIZE_POSITION = 3 THEN
           "PRIORITIZE_4" := 40;
           #PRIORITIZE_POSITION := 4;
       ELSIF #PRIORITIZE_POSITION = 4 THEN
           "PRIORITIZE_5" := 40;
           #PRIORITIZE_POSITION := 5;
       ELSIF #PRIORITIZE_POSITION = 5 THEN
           "PRIORITIZE_6" := 40;
           #PRIORITIZE_POSITION := 6;
       ELSIF #PRIORITIZE_POSITION = 6 THEN
           "PRIORITIZE_7" := 40;
           #PRIORITIZE_POSITION := 7;
       ELSIF #PRIORITIZE_POSITION = 7 THEN
           "PRIORITIZE_8" := 40;
           #PRIORITIZE_POSITION := 8;

           ;
       END_IF;
       ;
   END_IF;
   //F3 ĐI XUỐNG
   IF #F3_Down_Selected = TRUE THEN
       IF #PRIORITIZE_POSITION = 0 THEN
           "PRIORITIZE_1" := 30;
           #PRIORITIZE_POSITION := 1;
       ELSIF #PRIORITIZE_POSITION = 1 THEN
           "PRIORITIZE_2" := 30;
           #PRIORITIZE_POSITION := 2;
       ELSIF #PRIORITIZE_POSITION = 2 THEN
           "PRIORITIZE_3" := 30;
           #PRIORITIZE_POSITION := 3;
       ELSIF #PRIORITIZE_POSITION = 3 THEN
           "PRIORITIZE_4" := 30;
           #PRIORITIZE_POSITION := 4;
       ELSIF #PRIORITIZE_POSITION = 4 THEN
           "PRIORITIZE_5" := 30;
           #PRIORITIZE_POSITION := 5;
       ELSIF #PRIORITIZE_POSITION = 5 THEN
           "PRIORITIZE_6" := 30;
           #PRIORITIZE_POSITION := 6;
       ELSIF #PRIORITIZE_POSITION = 6 THEN
           "PRIORITIZE_7" := 30;
           #PRIORITIZE_POSITION := 7;
       ELSIF #PRIORITIZE_POSITION = 7 THEN
           "PRIORITIZE_8" := 30;
           #PRIORITIZE_POSITION := 8;

           ;
       END_IF;
       ;
   END_IF;
   // F2 ĐI XUỐNG
   IF #F2_Down_Selected = TRUE THEN
       IF #PRIORITIZE_POSITION = 0 THEN
           "PRIORITIZE_1" := 20;
           #PRIORITIZE_POSITION := 1;
       ELSIF #PRIORITIZE_POSITION = 1 THEN
           "PRIORITIZE_2" := 20;
           #PRIORITIZE_POSITION := 2;
       ELSIF #PRIORITIZE_POSITION = 2 THEN
           "PRIORITIZE_3" := 20;
           #PRIORITIZE_POSITION := 3;
       ELSIF #PRIORITIZE_POSITION = 3 THEN
           "PRIORITIZE_4" := 20;
           #PRIORITIZE_POSITION := 4;
       ELSIF #PRIORITIZE_POSITION = 4 THEN
           "PRIORITIZE_5" := 20;
           #PRIORITIZE_POSITION := 5;
       ELSIF #PRIORITIZE_POSITION = 5 THEN
           "PRIORITIZE_6" := 20;
           #PRIORITIZE_POSITION := 6;
       ELSIF #PRIORITIZE_POSITION = 6 THEN
           "PRIORITIZE_7" := 20;
           #PRIORITIZE_POSITION := 7;
       ELSIF #PRIORITIZE_POSITION = 7 THEN
           "PRIORITIZE_8" := 20;
           #PRIORITIZE_POSITION := 8;

           ;
       END_IF;
       ;
   END_IF;


   // MOVE TO OUTPUT
   // 
   #PRI_1 := "PRIORITIZE_1";
   #PRI_2 := "PRIORITIZE_2";
   #PRI_3 := "PRIORITIZE_3";
   #PRI_4 := "PRIORITIZE_4";
   #PRI_5 := "PRIORITIZE_5";
   #PRI_6 := "PRIORITIZE_6";
   #PRI_7 := "PRIORITIZE_7";
   #PRI_8 := "PRIORITIZE_8";
END_FUNCTION

FUNCTION "3.FC_REMOVE_PRIOTIZE" : Void   // FC3, SCL
{ S7_Optimized_Access := 'TRUE' }
VERSION : 0.1
   VAR_INPUT
      Ext_Clear_Rq : Bool;   // Yêu cầu xóa ưu tiên từ FC12
      Up_Called_F2 : Bool;
      Up_Called_F3 : Bool;
      Up_Called_F4 : Bool;
      Down_Called_F1 : Bool;
      Down_Called_F2 : Bool;
      Down_Called_F3 : Bool;
      Uping_F2 : Bool;
      Uping_F3 : Bool;
      Uping_F4 : Bool;
      Downing_F1 : Bool;
      Downing_F2 : Bool;
      Downing_F3 : Bool;
   END_VAR
BEGIN
   // NẾU THANG MÁY ĐI LÊN GẶP LIMIT SWITCH MÀ PHÁT HIỆN CÓ Ô NHỚ ƯU TIÊN NÀO CHỨA MÃ ĐI LÊN THÌ XÓA NÓ ĐI
   // 
   // TẦNG 1
   //DOWING
   //
   IF "DB_Status".LS_F1 = 1 THEN
       IF "PRIORITIZE_1" = 11 THEN
           "PRIORITIZE_1" := 0;
       ELSIF "PRIORITIZE_2" = 11 THEN
           "PRIORITIZE_2" := 0;
       ELSIF "PRIORITIZE_3" = 11 THEN
           "PRIORITIZE_3" := 0;
       ELSIF "PRIORITIZE_4" = 11 THEN
           "PRIORITIZE_4" := 0;
       ELSIF "PRIORITIZE_5" = 11 THEN
           "PRIORITIZE_5" := 0;
       ELSIF "PRIORITIZE_6" = 11 THEN
           "PRIORITIZE_6" := 0;
       ELSIF "PRIORITIZE_7" = 11 THEN
           "PRIORITIZE_7" := 0;
       ELSIF "PRIORITIZE_8" = 11 THEN
           "PRIORITIZE_8" := 0;

           ;
       END_IF;
       ;
   END_IF;
   // TẦNG 2
   // UPPING
   IF #Uping_F2 = 1 THEN
       IF "PRIORITIZE_1" = 21 THEN
           "PRIORITIZE_1" := 0;
       ELSIF "PRIORITIZE_2" = 21 THEN
           "PRIORITIZE_2" := 0;
       ELSIF "PRIORITIZE_3" = 21 THEN
           "PRIORITIZE_3" := 0;
       ELSIF "PRIORITIZE_4" = 21 THEN
           "PRIORITIZE_4" := 0;
       ELSIF "PRIORITIZE_5" = 21 THEN
           "PRIORITIZE_5" := 0;
       ELSIF "PRIORITIZE_6" = 21 THEN
           "PRIORITIZE_6" := 0;
       ELSIF "PRIORITIZE_7" = 21 THEN
           "PRIORITIZE_7" := 0;
       ELSIF "PRIORITIZE_8" = 21 THEN
           "PRIORITIZE_8" := 0;

           ;
       END_IF;
       ;
   END_IF;
   //DOWING
   //
   IF #Downing_F2 = 1 THEN
       IF "PRIORITIZE_1" = 20 THEN
           "PRIORITIZE_1" := 0;
       ELSIF "PRIORITIZE_2" = 20 THEN
           "PRIORITIZE_2" := 0;
       ELSIF "PRIORITIZE_3" = 20 THEN
           "PRIORITIZE_3" := 0;
       ELSIF "PRIORITIZE_4" = 20 THEN
           "PRIORITIZE_4" := 0;
       ELSIF "PRIORITIZE_5" = 20 THEN
           "PRIORITIZE_5" := 0;
       ELSIF "PRIORITIZE_6" = 20 THEN
           "PRIORITIZE_6" := 0;
       ELSIF "PRIORITIZE_7" = 20 THEN
           "PRIORITIZE_7" := 0;
       ELSIF "PRIORITIZE_8" = 20 THEN
           "PRIORITIZE_8" := 0;

           ;
       END_IF;
       ;
   END_IF;
   // TẦNG 3
   // UPPING
   IF #Uping_F3 = 1 THEN
       IF "PRIORITIZE_1" = 31 THEN
           "PRIORITIZE_1" := 0;
       ELSIF "PRIORITIZE_2" = 31 THEN
           "PRIORITIZE_2" := 0;
       ELSIF "PRIORITIZE_3" = 31 THEN
           "PRIORITIZE_3" := 0;
       ELSIF "PRIORITIZE_4" = 31 THEN
           "PRIORITIZE_4" := 0;
       ELSIF "PRIORITIZE_5" = 31 THEN
           "PRIORITIZE_5" := 0;
       ELSIF "PRIORITIZE_6" = 31 THEN
           "PRIORITIZE_6" := 0;
       ELSIF "PRIORITIZE_7" = 31 THEN
           "PRIORITIZE_7" := 0;
       ELSIF "PRIORITIZE_8" = 31 THEN
           "PRIORITIZE_8" := 0;

           ;
       END_IF;
       ;
   END_IF;
   //DOWING
   //
   IF #Downing_F3 = 1 THEN
       IF "PRIORITIZE_1" = 30 THEN
           "PRIORITIZE_1" := 0;
       ELSIF "PRIORITIZE_2" = 30 THEN
           "PRIORITIZE_2" := 0;
       ELSIF "PRIORITIZE_3" = 30 THEN
           "PRIORITIZE_3" := 0;
       ELSIF "PRIORITIZE_4" = 30 THEN
           "PRIORITIZE_4" := 0;
       ELSIF "PRIORITIZE_5" = 30 THEN
           "PRIORITIZE_5" := 0;
       ELSIF "PRIORITIZE_6" = 30 THEN
           "PRIORITIZE_6" := 0;
       ELSIF "PRIORITIZE_7" = 30 THEN
           "PRIORITIZE_7" := 0;
       ELSIF "PRIORITIZE_8" = 30 THEN
           "PRIORITIZE_8" := 0;
           ;
       END_IF;
       ;
   END_IF;
   // TẦNG 4
   // UPPING
   IF #Uping_F4 = 1 THEN
       IF "PRIORITIZE_1" = 41 THEN
           "PRIORITIZE_1" := 0;
       ELSIF "PRIORITIZE_2" = 41 THEN
           "PRIORITIZE_2" := 0;
       ELSIF "PRIORITIZE_3" = 41 THEN
           "PRIORITIZE_3" := 0;
       ELSIF "PRIORITIZE_4" = 41 THEN
           "PRIORITIZE_4" := 0;
       ELSIF "PRIORITIZE_5" = 41 THEN
           "PRIORITIZE_5" := 0;
       ELSIF "PRIORITIZE_6" = 41 THEN
           "PRIORITIZE_6" := 0;
       ELSIF "PRIORITIZE_7" = 41 THEN
           "PRIORITIZE_7" := 0;
       ELSIF "PRIORITIZE_8" = 41 THEN
           "PRIORITIZE_8" := 0;
       ELSIF "PRIORITIZE_9" = 41 THEN
           "PRIORITIZE_9" := 0;
       ELSIF "PRIORITIZE_10" = 41 THEN
           "PRIORITIZE_10" := 0;
       ELSIF "PRIORITIZE_11" = 41 THEN
           "PRIORITIZE_11" := 0;
       ELSIF "PRIORITIZE_12" = 41 THEN
           "PRIORITIZE_12" := 0;
           ;
       END_IF;
       ;
   END_IF;
   //DOWING
   //
   IF "DB_Status".LS_F4 = 1 THEN
       IF "PRIORITIZE_1" = 40 THEN
           "PRIORITIZE_1" := 0;
       ELSIF "PRIORITIZE_2" = 40 THEN
           "PRIORITIZE_2" := 0;
       ELSIF "PRIORITIZE_3" = 40 THEN
           "PRIORITIZE_3" := 0;
       ELSIF "PRIORITIZE_4" = 40 THEN
           "PRIORITIZE_4" := 0;
       ELSIF "PRIORITIZE_5" = 40 THEN
           "PRIORITIZE_5" := 0;
       ELSIF "PRIORITIZE_6" = 40 THEN
           "PRIORITIZE_6" := 0;
       ELSIF "PRIORITIZE_7" = 40 THEN
           "PRIORITIZE_7" := 0;
       ELSIF "PRIORITIZE_8" = 40 THEN
           "PRIORITIZE_8" := 0;

           ;
       END_IF;
       ;
   END_IF;







   // YÊU CẦU XÓA ƯU TIÊN TỪ FC12
   // 
   // F1 UP
   IF #Ext_Clear_Rq = 1 & #Down_Called_F1 = 1 & #Downing_F1 = 1 THEN
       IF "PRIORITIZE_1" = 10 THEN
           "PRIORITIZE_1" := 0;
       ELSIF "PRIORITIZE_2" = 10 THEN
           "PRIORITIZE_2" := 0;
       ELSIF "PRIORITIZE_3" = 10 THEN
           "PRIORITIZE_3" := 0;
       ELSIF "PRIORITIZE_4" = 10 THEN
           "PRIORITIZE_4" := 0;
       ELSIF "PRIORITIZE_5" = 10 THEN
           "PRIORITIZE_5" := 0;
       ELSIF "PRIORITIZE_6" = 10 THEN
           "PRIORITIZE_6" := 0;
       ELSIF "PRIORITIZE_7" = 10 THEN
           "PRIORITIZE_7" := 0;
       ELSIF "PRIORITIZE_8" = 10 THEN
           "PRIORITIZE_8" := 0;

           ;
       END_IF;
       ;
   END_IF;

   // F2 UP
   IF #Ext_Clear_Rq = 1 & #Up_Called_F2 = 1 & #Downing_F2 = 1 THEN
       IF "PRIORITIZE_1" = 21 THEN
           "PRIORITIZE_1" := 0;
       ELSIF "PRIORITIZE_2" = 21 THEN
           "PRIORITIZE_2" := 0;
       ELSIF "PRIORITIZE_3" = 21 THEN
           "PRIORITIZE_3" := 0;
       ELSIF "PRIORITIZE_4" = 21 THEN
           "PRIORITIZE_4" := 0;
       ELSIF "PRIORITIZE_5" = 21 THEN
           "PRIORITIZE_5" := 0;
       ELSIF "PRIORITIZE_6" = 21 THEN
           "PRIORITIZE_6" := 0;
       ELSIF "PRIORITIZE_7" = 21 THEN
           "PRIORITIZE_7" := 0;
       ELSIF "PRIORITIZE_8" = 21 THEN
           "PRIORITIZE_8" := 0;

           ;
       END_IF;
       ;
   END_IF;

   // F2 DOWN
   IF #Ext_Clear_Rq = 1 & #Down_Called_F2 = 1 & #Uping_F2 = 1 THEN
       IF "PRIORITIZE_1" = 20 THEN
           "PRIORITIZE_1" := 0;
       ELSIF "PRIORITIZE_2" = 20 THEN
           "PRIORITIZE_2" := 0;
       ELSIF "PRIORITIZE_3" = 20 THEN
           "PRIORITIZE_3" := 0;
       ELSIF "PRIORITIZE_4" = 20 THEN
           "PRIORITIZE_4" := 0;
       ELSIF "PRIORITIZE_5" = 20 THEN
           "PRIORITIZE_5" := 0;
       ELSIF "PRIORITIZE_6" = 20 THEN
           "PRIORITIZE_6" := 0;
       ELSIF "PRIORITIZE_7" = 20 THEN
           "PRIORITIZE_7" := 0;
       ELSIF "PRIORITIZE_8" = 20 THEN
           "PRIORITIZE_8" := 0;

           ;
       END_IF;
       ;
   END_IF;

   // F3 UP
   IF #Ext_Clear_Rq = 1 & #Up_Called_F3 = 1 & #Downing_F3 = 1 THEN
       IF "PRIORITIZE_1" = 31 THEN
           "PRIORITIZE_1" := 0;
       ELSIF "PRIORITIZE_2" = 31 THEN
           "PRIORITIZE_2" := 0;
       ELSIF "PRIORITIZE_3" = 31 THEN
           "PRIORITIZE_3" := 0;
       ELSIF "PRIORITIZE_4" = 31 THEN
           "PRIORITIZE_4" := 0;
       ELSIF "PRIORITIZE_5" = 31 THEN
           "PRIORITIZE_5" := 0;
       ELSIF "PRIORITIZE_6" = 31 THEN
           "PRIORITIZE_6" := 0;
       ELSIF "PRIORITIZE_7" = 31 THEN
           "PRIORITIZE_7" := 0;
       ELSIF "PRIORITIZE_8" = 31 THEN
           "PRIORITIZE_8" := 0;

           ;
       END_IF;
       ;
   END_IF;

   // F3 DOWN
   IF #Ext_Clear_Rq = 1 & #Down_Called_F3 = 1 & #Uping_F3 = 1 THEN
       IF "PRIORITIZE_1" = 30 THEN
           "PRIORITIZE_1" := 0;
       ELSIF "PRIORITIZE_2" = 30 THEN
           "PRIORITIZE_2" := 0;
       ELSIF "PRIORITIZE_3" = 30 THEN
           "PRIORITIZE_3" := 0;
       ELSIF "PRIORITIZE_4" = 30 THEN
           "PRIORITIZE_4" := 0;
       ELSIF "PRIORITIZE_5" = 30 THEN
           "PRIORITIZE_5" := 0;
       ELSIF "PRIORITIZE_6" = 30 THEN
           "PRIORITIZE_6" := 0;
       ELSIF "PRIORITIZE_7" = 30 THEN
           "PRIORITIZE_7" := 0;
       ELSIF "PRIORITIZE_8" = 30 THEN
           "PRIORITIZE_8" := 0;

           ;
       END_IF;
       ;
   END_IF;



   // F4 up
   IF #Ext_Clear_Rq = 1 & #Up_Called_F4 = 1 & #Uping_F4 = 1 THEN 
       IF "PRIORITIZE_1" = 40 THEN
           "PRIORITIZE_1" := 0;
       ELSIF "PRIORITIZE_2" = 40 THEN
           "PRIORITIZE_2" := 0;
       ELSIF "PRIORITIZE_3" = 40 THEN
           "PRIORITIZE_3" := 0;
       ELSIF "PRIORITIZE_4" = 40 THEN
           "PRIORITIZE_4" := 0;
       ELSIF "PRIORITIZE_5" = 40 THEN
           "PRIORITIZE_5" := 0;
       ELSIF "PRIORITIZE_6" = 40 THEN
           "PRIORITIZE_6" := 0;
       ELSIF "PRIORITIZE_7" = 40 THEN
           "PRIORITIZE_7" := 0;
       ELSIF "PRIORITIZE_8" = 40 THEN
           "PRIORITIZE_8" := 0;
       ELSIF "PRIORITIZE_9" = 40 THEN
           "PRIORITIZE_9" := 0;
       ELSIF "PRIORITIZE_10" = 40 THEN
           "PRIORITIZE_10" := 0;
       ELSIF "PRIORITIZE_11" = 40 THEN
           "PRIORITIZE_11" := 0;
       ELSIF "PRIORITIZE_12" = 40 THEN
           "PRIORITIZE_12" := 0;
           ;
       END_IF;
       ;
   END_IF;
END_FUNCTION

FUNCTION "4.FC_CABINET_STATUS" : Void   // FC4, LAD
{ S7_Optimized_Access := 'TRUE' }
VERSION : 0.1
// BLOCK TRẠNG THÁI VÀ VỊ TRÍ CỦA BUỒNG THANG
   VAR_TEMP   // added for the SCL form of the ladder/FBD networks
      _w1 : Bool;
      _w2 : Bool;
   END_VAR
BEGIN

REGION Network 1: BUỒNG THANG ĐANG XUỐNG TẦNG 1
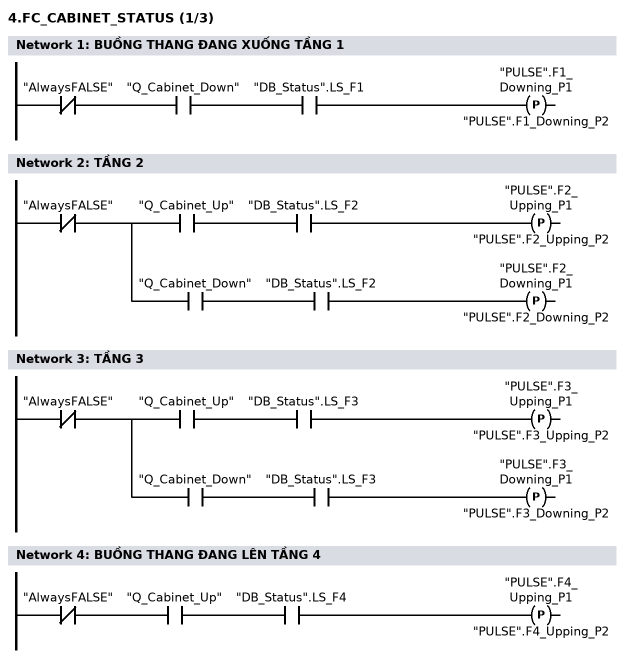
   #_w1 := NOT "AlwaysFALSE" AND "Q_Cabinet_Down" AND "DB_Status".LS_F1;
   "PULSE".F1_Downing_P1 := #_w1 AND NOT "PULSE".F1_Downing_P2;   // rising edge
   "PULSE".F1_Downing_P2 := #_w1;
END_REGION

REGION Network 2: TẦNG 2
   #_w1 := NOT "AlwaysFALSE" AND "Q_Cabinet_Up" AND "DB_Status".LS_F2;
   "PULSE".F2_Upping_P1 := #_w1 AND NOT "PULSE".F2_Upping_P2;   // rising edge
   "PULSE".F2_Upping_P2 := #_w1;
   #_w2 := NOT "AlwaysFALSE" AND "Q_Cabinet_Down" AND "DB_Status".LS_F2;
   "PULSE".F2_Downing_P1 := #_w2 AND NOT "PULSE".F2_Downing_P2;   // rising edge
   "PULSE".F2_Downing_P2 := #_w2;
END_REGION

REGION Network 3: TẦNG 3
   #_w1 := NOT "AlwaysFALSE" AND "Q_Cabinet_Up" AND "DB_Status".LS_F3;
   "PULSE".F3_Upping_P1 := #_w1 AND NOT "PULSE".F3_Upping_P2;   // rising edge
   "PULSE".F3_Upping_P2 := #_w1;
   #_w2 := NOT "AlwaysFALSE" AND "Q_Cabinet_Down" AND "DB_Status".LS_F3;
   "PULSE".F3_Downing_P1 := #_w2 AND NOT "PULSE".F3_Downing_P2;   // rising edge
   "PULSE".F3_Downing_P2 := #_w2;
END_REGION

REGION Network 4: BUỒNG THANG ĐANG LÊN TẦNG 4
   #_w1 := NOT "AlwaysFALSE" AND "Q_Cabinet_Up" AND "DB_Status".LS_F4;
   "PULSE".F4_Upping_P1 := #_w1 AND NOT "PULSE".F4_Upping_P2;   // rising edge
   "PULSE".F4_Upping_P2 := #_w1;
END_REGION

REGION Network 5: HIEN THI TRANG THAI 2S
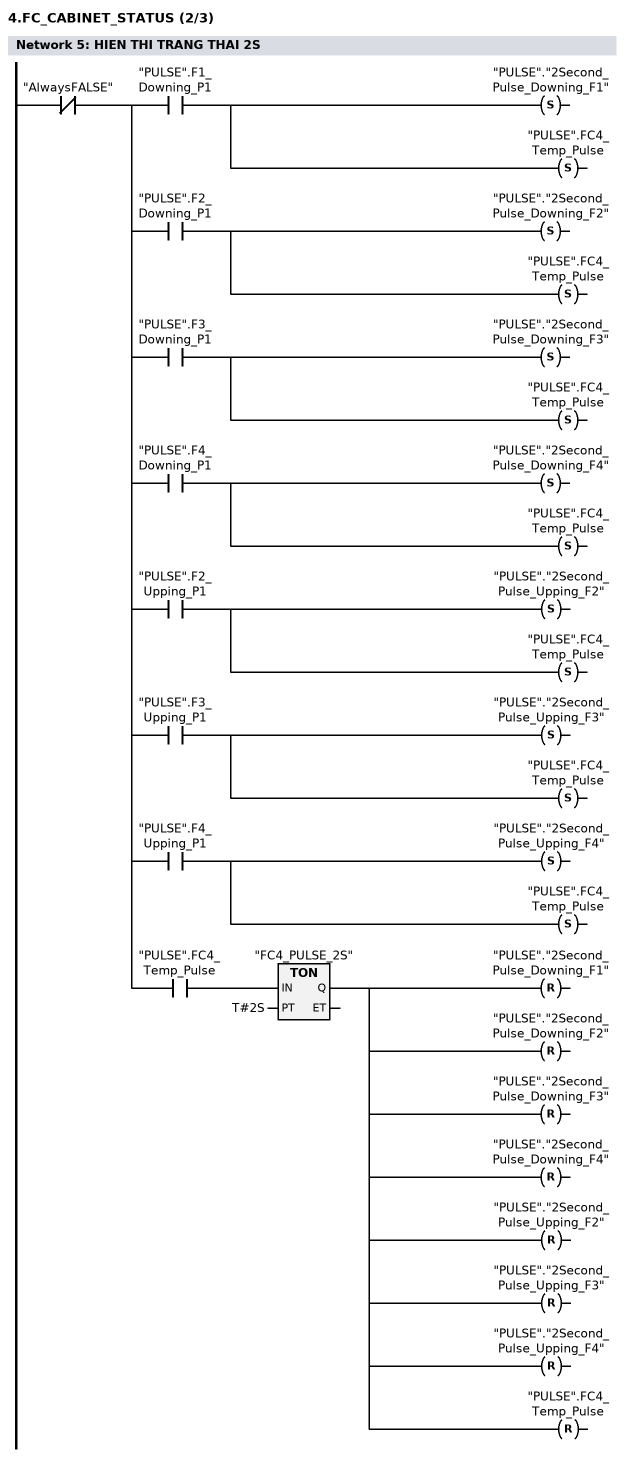
   IF NOT "AlwaysFALSE" AND "PULSE".F1_Downing_P1 THEN
       "PULSE"."2Second_Pulse_Downing_F1" := TRUE;
       "PULSE".FC4_Temp_Pulse := TRUE;
   END_IF;
   IF NOT "AlwaysFALSE" AND "PULSE".F2_Downing_P1 THEN
       "PULSE"."2Second_Pulse_Downing_F2" := TRUE;
       "PULSE".FC4_Temp_Pulse := TRUE;
   END_IF;
   IF NOT "AlwaysFALSE" AND "PULSE".F3_Downing_P1 THEN
       "PULSE"."2Second_Pulse_Downing_F3" := TRUE;
       "PULSE".FC4_Temp_Pulse := TRUE;
   END_IF;
   IF NOT "AlwaysFALSE" AND "PULSE".F4_Downing_P1 THEN
       "PULSE"."2Second_Pulse_Downing_F4" := TRUE;
       "PULSE".FC4_Temp_Pulse := TRUE;
   END_IF;
   IF NOT "AlwaysFALSE" AND "PULSE".F2_Upping_P1 THEN
       "PULSE"."2Second_Pulse_Upping_F2" := TRUE;
       "PULSE".FC4_Temp_Pulse := TRUE;
   END_IF;
   IF NOT "AlwaysFALSE" AND "PULSE".F3_Upping_P1 THEN
       "PULSE"."2Second_Pulse_Upping_F3" := TRUE;
       "PULSE".FC4_Temp_Pulse := TRUE;
   END_IF;
   IF NOT "AlwaysFALSE" AND "PULSE".F4_Upping_P1 THEN
       "PULSE"."2Second_Pulse_Upping_F4" := TRUE;
       "PULSE".FC4_Temp_Pulse := TRUE;
   END_IF;
   "FC4_PULSE_2S".TON(IN := NOT "AlwaysFALSE" AND "PULSE".FC4_Temp_Pulse, PT := T#2S);
   IF "FC4_PULSE_2S".Q THEN
       "PULSE"."2Second_Pulse_Downing_F1" := FALSE;
       "PULSE"."2Second_Pulse_Downing_F2" := FALSE;
       "PULSE"."2Second_Pulse_Downing_F3" := FALSE;
       "PULSE"."2Second_Pulse_Downing_F4" := FALSE;
       "PULSE"."2Second_Pulse_Upping_F2" := FALSE;
       "PULSE"."2Second_Pulse_Upping_F3" := FALSE;
       "PULSE"."2Second_Pulse_Upping_F4" := FALSE;
       "PULSE".FC4_Temp_Pulse := FALSE;
   END_IF;
END_REGION

REGION Network 6: HIỂN THỊ VỊ TRÍ TẦNG
   // 1 = TẦNG 1, ... 6 = TẦNG 6
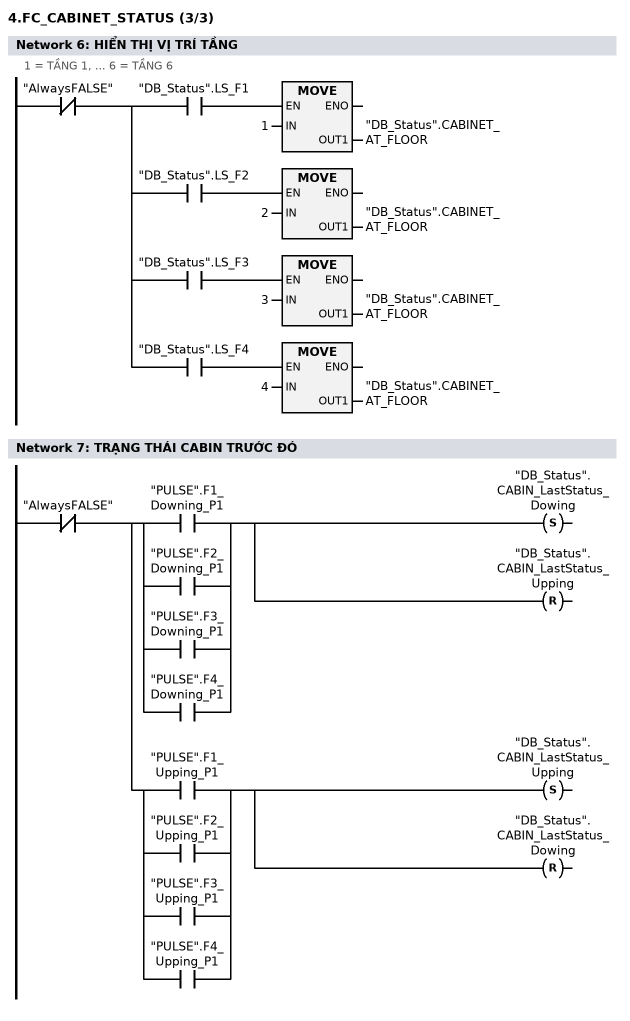
   RUNG wire#powerrail
      I_Contact( "AlwaysFALSE" )
      wire#w1
      Contact( "DB_Status".LS_F1 )
      Move(in := 1, out1 => "DB_Status".CABINET_AT_FLOOR)
   END_RUNG
   RUNG wire#w1
      Contact( "DB_Status".LS_F2 )
      Move(in := 2, out1 => "DB_Status".CABINET_AT_FLOOR)
   END_RUNG
   RUNG wire#w1
      Contact( "DB_Status".LS_F3 )
      Move(in := 3, out1 => "DB_Status".CABINET_AT_FLOOR)
   END_RUNG
   RUNG wire#w1
      Contact( "DB_Status".LS_F4 )
      Move(in := 4, out1 => "DB_Status".CABINET_AT_FLOOR)
   END_RUNG
   // the same network as SCL:
   IF NOT "AlwaysFALSE" AND "DB_Status".LS_F1 THEN "DB_Status".CABINET_AT_FLOOR := 1; END_IF;
   IF NOT "AlwaysFALSE" AND "DB_Status".LS_F2 THEN "DB_Status".CABINET_AT_FLOOR := 2; END_IF;
   IF NOT "AlwaysFALSE" AND "DB_Status".LS_F3 THEN "DB_Status".CABINET_AT_FLOOR := 3; END_IF;
   IF NOT "AlwaysFALSE" AND "DB_Status".LS_F4 THEN "DB_Status".CABINET_AT_FLOOR := 4; END_IF;
END_REGION

REGION Network 7: TRẠNG THÁI CABIN TRƯỚC ĐÓ
   RUNG wire#powerrail
      I_Contact( "AlwaysFALSE" )
      wire#w1
      Contact( "PULSE".F1_Downing_P1 )
      wire#w2
      S_Coil( "DB_Status".CABIN_LastStatus_Dowing )
   END_RUNG
   RUNG wire#w1
      Contact( "PULSE".F2_Downing_P1 )
   END_RUNG wire#w2
   RUNG wire#w1
      Contact( "PULSE".F3_Downing_P1 )
   END_RUNG wire#w2
   RUNG wire#w1
      Contact( "PULSE".F4_Downing_P1 )
   END_RUNG wire#w2
   RUNG wire#w2
      R_Coil( "DB_Status".CABIN_LastStatus_Upping )
   END_RUNG
   RUNG wire#w1
      Contact( "PULSE".F1_Upping_P1 )
      wire#w3
      S_Coil( "DB_Status".CABIN_LastStatus_Upping )
   END_RUNG
   RUNG wire#w1
      Contact( "PULSE".F2_Upping_P1 )
   END_RUNG wire#w3
   RUNG wire#w1
      Contact( "PULSE".F3_Upping_P1 )
   END_RUNG wire#w3
   RUNG wire#w1
      Contact( "PULSE".F4_Upping_P1 )
   END_RUNG wire#w3
   RUNG wire#w3
      R_Coil( "DB_Status".CABIN_LastStatus_Dowing )
   END_RUNG
   // the same network as SCL:
   IF NOT "AlwaysFALSE" AND ("PULSE".F1_Downing_P1 OR "PULSE".F2_Downing_P1 OR "PULSE".F3_Downing_P1 OR "PULSE".F4_Downing_P1) THEN
       "DB_Status".CABIN_LastStatus_Dowing := TRUE;
       "DB_Status".CABIN_LastStatus_Upping := FALSE;
   END_IF;
   IF NOT "AlwaysFALSE" AND ("PULSE".F1_Upping_P1 OR "PULSE".F2_Upping_P1 OR "PULSE".F3_Upping_P1 OR "PULSE".F4_Upping_P1) THEN
       "DB_Status".CABIN_LastStatus_Upping := TRUE;
       "DB_Status".CABIN_LastStatus_Dowing := FALSE;
   END_IF;
END_REGION
END_FUNCTION

FUNCTION "5.FC_CABINET_CONTROL" : Void   // FC5, LAD
{ S7_Optimized_Access := 'TRUE' }
VERSION : 0.1
   VAR_INPUT
      Ext_Stop_Rq : Bool;   // Yêu cầu dừng ca bin
      LS_Door_Opened : Bool;   // Limit switch cửa đóng
      LS_Door_Closed : Bool;   // Limit switch cửa mở
      Pls_Door_Lock : Bool;   // Cửa đóng 3s thì lock để di chuyển buồng thang
      Upping_F2 : Bool;   // Buồng thang lên đến tầng 2
      Upping_F3 : Bool;   // Buồng thang lên đến tầng 3
      Upping_F4 : Bool;   // Buồng thang lên đến tầng 4
      Upping_F5 : Bool;   // Buồng thang lên đến tầng 5
      Upping_F6 : Bool;   // Buồng thang lên đến tầng 6
      Downing_F1 : Bool;   // Buồng thang về đến tầng 1
      Downing_F2 : Bool;   // Buồng thang về đến tầng 2
      Downing_F3 : Bool;   // Buồng thang về đến tầng 3
      Downing_F4 : Bool;   // Buồng thang về đến tầng 4
      Downing_F5 : Bool;   // Buồng thang về đến tầng 5
      Next_Floor : SInt;   // Tầng kế tiếp cần đi tới
   END_VAR
   VAR_OUTPUT
      OR_Cabinet_Up : Bool;
      OR_Cabinet_Down : Bool;
   END_VAR
BEGIN

REGION Network 1: THANG ĐANG Ở TẦNG 1
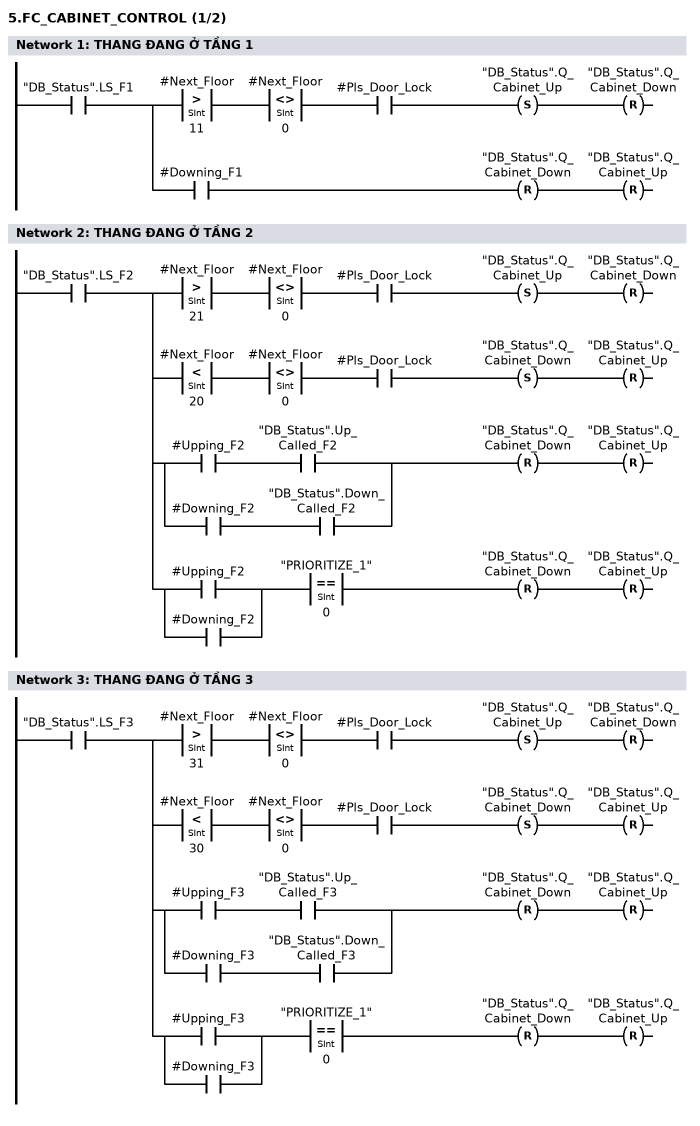
   RUNG wire#powerrail
      Contact( "DB_Status".LS_F1 )
      wire#w1
      { S7_Templates := "SrcType := SInt" } GT_Contact(in1 := #Next_Floor, in2 := 11)
      { S7_Templates := "SrcType := SInt" } NE_Contact(in1 := #Next_Floor, in2 := 0)
      Contact( #Pls_Door_Lock )
      S_Coil( "DB_Status".Q_Cabinet_Up )
      R_Coil( "DB_Status".Q_Cabinet_Down )
   END_RUNG
   RUNG wire#w1
      Contact( #Downing_F1 )
      R_Coil( "DB_Status".Q_Cabinet_Down )
      R_Coil( "DB_Status".Q_Cabinet_Up )
   END_RUNG
   // the same network as SCL:
   IF "DB_Status".LS_F1 AND (#Next_Floor > 11) AND (#Next_Floor <> 0) AND #Pls_Door_Lock THEN
       "DB_Status".Q_Cabinet_Up := TRUE;
       "DB_Status".Q_Cabinet_Down := FALSE;
   END_IF;
   IF "DB_Status".LS_F1 AND #Downing_F1 THEN
       "DB_Status".Q_Cabinet_Down := FALSE;
       "DB_Status".Q_Cabinet_Up := FALSE;
   END_IF;
END_REGION

REGION Network 2: THANG ĐANG Ở TẦNG 2
   RUNG wire#powerrail
      Contact( "DB_Status".LS_F2 )
      wire#w1
      { S7_Templates := "SrcType := SInt" } GT_Contact(in1 := #Next_Floor, in2 := 21)
      { S7_Templates := "SrcType := SInt" } NE_Contact(in1 := #Next_Floor, in2 := 0)
      Contact( #Pls_Door_Lock )
      S_Coil( "DB_Status".Q_Cabinet_Up )
      R_Coil( "DB_Status".Q_Cabinet_Down )
   END_RUNG
   RUNG wire#w1
      { S7_Templates := "SrcType := SInt" } LT_Contact(in1 := #Next_Floor, in2 := 20)
      { S7_Templates := "SrcType := SInt" } NE_Contact(in1 := #Next_Floor, in2 := 0)
      Contact( #Pls_Door_Lock )
      S_Coil( "DB_Status".Q_Cabinet_Down )
      R_Coil( "DB_Status".Q_Cabinet_Up )
   END_RUNG
   RUNG wire#w1
      Contact( #Upping_F2 )
      Contact( "DB_Status".Up_Called_F2 )
      wire#w2
      R_Coil( "DB_Status".Q_Cabinet_Down )
      R_Coil( "DB_Status".Q_Cabinet_Up )
   END_RUNG
   RUNG wire#w1
      Contact( #Downing_F2 )
      Contact( "DB_Status".Down_Called_F2 )
   END_RUNG wire#w2
   RUNG wire#w1
      Contact( #Upping_F2 )
      wire#w3
      { S7_Templates := "SrcType := SInt" } EQ_Contact(in1 := "PRIORITIZE_1", in2 := 0)
      R_Coil( "DB_Status".Q_Cabinet_Down )
      R_Coil( "DB_Status".Q_Cabinet_Up )
   END_RUNG
   RUNG wire#w1
      Contact( #Downing_F2 )
   END_RUNG wire#w3
   // the same network as SCL:
   IF "DB_Status".LS_F2 AND (#Next_Floor > 21) AND (#Next_Floor <> 0) AND #Pls_Door_Lock THEN
       "DB_Status".Q_Cabinet_Up := TRUE;
       "DB_Status".Q_Cabinet_Down := FALSE;
   END_IF;
   IF "DB_Status".LS_F2 AND (#Next_Floor < 20) AND (#Next_Floor <> 0) AND #Pls_Door_Lock THEN
       "DB_Status".Q_Cabinet_Down := TRUE;
       "DB_Status".Q_Cabinet_Up := FALSE;
   END_IF;
   IF "DB_Status".LS_F2 AND ((#Upping_F2 AND "DB_Status".Up_Called_F2) OR (#Downing_F2 AND "DB_Status".Down_Called_F2)) THEN
       "DB_Status".Q_Cabinet_Down := FALSE;
       "DB_Status".Q_Cabinet_Up := FALSE;
   END_IF;
   IF "DB_Status".LS_F2 AND (#Upping_F2 OR #Downing_F2) AND ("PRIORITIZE_1" = 0) THEN
       "DB_Status".Q_Cabinet_Down := FALSE;
       "DB_Status".Q_Cabinet_Up := FALSE;
   END_IF;
END_REGION

REGION Network 3: THANG ĐANG Ở TẦNG 3
   RUNG wire#powerrail
      Contact( "DB_Status".LS_F3 )
      wire#w1
      { S7_Templates := "SrcType := SInt" } GT_Contact(in1 := #Next_Floor, in2 := 31)
      { S7_Templates := "SrcType := SInt" } NE_Contact(in1 := #Next_Floor, in2 := 0)
      Contact( #Pls_Door_Lock )
      S_Coil( "DB_Status".Q_Cabinet_Up )
      R_Coil( "DB_Status".Q_Cabinet_Down )
   END_RUNG
   RUNG wire#w1
      { S7_Templates := "SrcType := SInt" } LT_Contact(in1 := #Next_Floor, in2 := 30)
      { S7_Templates := "SrcType := SInt" } NE_Contact(in1 := #Next_Floor, in2 := 0)
      Contact( #Pls_Door_Lock )
      S_Coil( "DB_Status".Q_Cabinet_Down )
      R_Coil( "DB_Status".Q_Cabinet_Up )
   END_RUNG
   RUNG wire#w1
      Contact( #Upping_F3 )
      Contact( "DB_Status".Up_Called_F3 )
      wire#w2
      R_Coil( "DB_Status".Q_Cabinet_Down )
      R_Coil( "DB_Status".Q_Cabinet_Up )
   END_RUNG
   RUNG wire#w1
      Contact( #Downing_F3 )
      Contact( "DB_Status".Down_Called_F3 )
   END_RUNG wire#w2
   RUNG wire#w1
      Contact( #Upping_F3 )
      wire#w3
      { S7_Templates := "SrcType := SInt" } EQ_Contact(in1 := "PRIORITIZE_1", in2 := 0)
      R_Coil( "DB_Status".Q_Cabinet_Down )
      R_Coil( "DB_Status".Q_Cabinet_Up )
   END_RUNG
   RUNG wire#w1
      Contact( #Downing_F3 )
   END_RUNG wire#w3
   // the same network as SCL:
   IF "DB_Status".LS_F3 AND (#Next_Floor > 31) AND (#Next_Floor <> 0) AND #Pls_Door_Lock THEN
       "DB_Status".Q_Cabinet_Up := TRUE;
       "DB_Status".Q_Cabinet_Down := FALSE;
   END_IF;
   IF "DB_Status".LS_F3 AND (#Next_Floor < 30) AND (#Next_Floor <> 0) AND #Pls_Door_Lock THEN
       "DB_Status".Q_Cabinet_Down := TRUE;
       "DB_Status".Q_Cabinet_Up := FALSE;
   END_IF;
   IF "DB_Status".LS_F3 AND ((#Upping_F3 AND "DB_Status".Up_Called_F3) OR (#Downing_F3 AND "DB_Status".Down_Called_F3)) THEN
       "DB_Status".Q_Cabinet_Down := FALSE;
       "DB_Status".Q_Cabinet_Up := FALSE;
   END_IF;
   IF "DB_Status".LS_F3 AND (#Upping_F3 OR #Downing_F3) AND ("PRIORITIZE_1" = 0) THEN
       "DB_Status".Q_Cabinet_Down := FALSE;
       "DB_Status".Q_Cabinet_Up := FALSE;
   END_IF;
END_REGION

REGION Network 4: THANG ĐANG Ở TẦNG 4
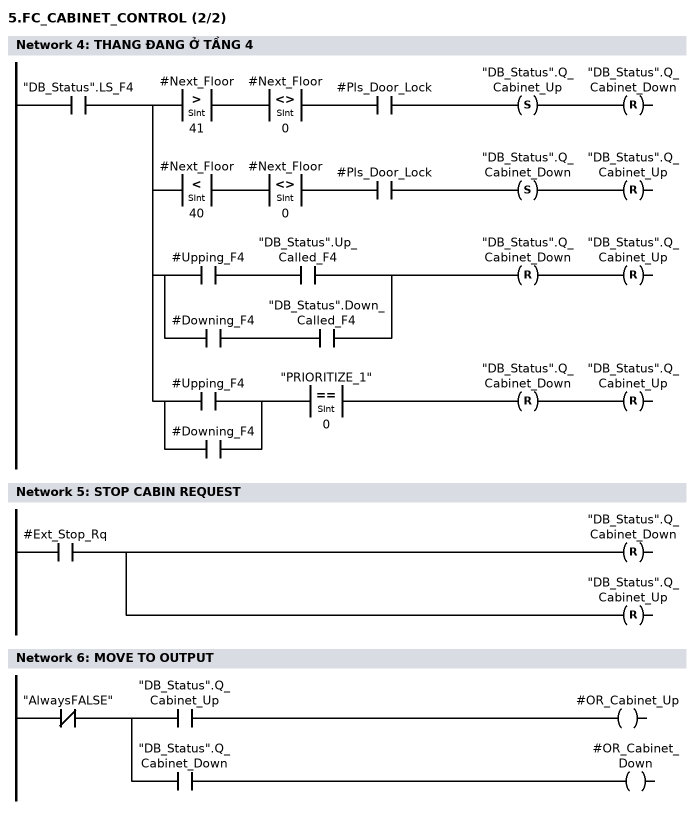
   RUNG wire#powerrail
      Contact( "DB_Status".LS_F4 )
      wire#w1
      { S7_Templates := "SrcType := SInt" } GT_Contact(in1 := #Next_Floor, in2 := 41)
      { S7_Templates := "SrcType := SInt" } NE_Contact(in1 := #Next_Floor, in2 := 0)
      Contact( #Pls_Door_Lock )
      S_Coil( "DB_Status".Q_Cabinet_Up )
      R_Coil( "DB_Status".Q_Cabinet_Down )
   END_RUNG
   RUNG wire#w1
      { S7_Templates := "SrcType := SInt" } LT_Contact(in1 := #Next_Floor, in2 := 40)
      { S7_Templates := "SrcType := SInt" } NE_Contact(in1 := #Next_Floor, in2 := 0)
      Contact( #Pls_Door_Lock )
      S_Coil( "DB_Status".Q_Cabinet_Down )
      R_Coil( "DB_Status".Q_Cabinet_Up )
   END_RUNG
   RUNG wire#w1
      Contact( #Upping_F4 )
      Contact( "DB_Status".Up_Called_F4 )
      wire#w2
      R_Coil( "DB_Status".Q_Cabinet_Down )
      R_Coil( "DB_Status".Q_Cabinet_Up )
   END_RUNG
   RUNG wire#w1
      Contact( #Downing_F4 )
      Contact( "DB_Status".Down_Called_F4 )
   END_RUNG wire#w2
   RUNG wire#w1
      Contact( #Upping_F4 )
      wire#w3
      { S7_Templates := "SrcType := SInt" } EQ_Contact(in1 := "PRIORITIZE_1", in2 := 0)
      R_Coil( "DB_Status".Q_Cabinet_Down )
      R_Coil( "DB_Status".Q_Cabinet_Up )
   END_RUNG
   RUNG wire#w1
      Contact( #Downing_F4 )
   END_RUNG wire#w3
   // the same network as SCL:
   IF "DB_Status".LS_F4 AND (#Next_Floor > 41) AND (#Next_Floor <> 0) AND #Pls_Door_Lock THEN
       "DB_Status".Q_Cabinet_Up := TRUE;
       "DB_Status".Q_Cabinet_Down := FALSE;
   END_IF;
   IF "DB_Status".LS_F4 AND (#Next_Floor < 40) AND (#Next_Floor <> 0) AND #Pls_Door_Lock THEN
       "DB_Status".Q_Cabinet_Down := TRUE;
       "DB_Status".Q_Cabinet_Up := FALSE;
   END_IF;
   IF "DB_Status".LS_F4 AND ((#Upping_F4 AND "DB_Status".Up_Called_F4) OR (#Downing_F4 AND "DB_Status".Down_Called_F4)) THEN
       "DB_Status".Q_Cabinet_Down := FALSE;
       "DB_Status".Q_Cabinet_Up := FALSE;
   END_IF;
   IF "DB_Status".LS_F4 AND (#Upping_F4 OR #Downing_F4) AND ("PRIORITIZE_1" = 0) THEN
       "DB_Status".Q_Cabinet_Down := FALSE;
       "DB_Status".Q_Cabinet_Up := FALSE;
   END_IF;
END_REGION

REGION Network 5: STOP CABIN REQUEST
   RUNG wire#powerrail
      Contact( #Ext_Stop_Rq )
      wire#w1
      R_Coil( "DB_Status".Q_Cabinet_Down )
   END_RUNG
   RUNG wire#w1
      R_Coil( "DB_Status".Q_Cabinet_Up )
   END_RUNG
   // the same network as SCL:
   IF #Ext_Stop_Rq THEN
       "DB_Status".Q_Cabinet_Down := FALSE;
       "DB_Status".Q_Cabinet_Up := FALSE;
   END_IF;
END_REGION

REGION Network 6: MOVE TO OUTPUT
   RUNG wire#powerrail
      I_Contact( "AlwaysFALSE" )
      wire#w1
      Contact( "DB_Status".Q_Cabinet_Up )
      Coil( #OR_Cabinet_Up )
   END_RUNG
   RUNG wire#w1
      Contact( "DB_Status".Q_Cabinet_Down )
      Coil( #OR_Cabinet_Down )
   END_RUNG
   // the same network as SCL:
   #OR_Cabinet_Up := NOT "AlwaysFALSE" AND "DB_Status".Q_Cabinet_Up;
   #OR_Cabinet_Down := NOT "AlwaysFALSE" AND "DB_Status".Q_Cabinet_Down;
END_REGION
END_FUNCTION

FUNCTION "6.FC_FLOOR_CALL" : Void   // FC6, SCL
{ S7_Optimized_Access := 'TRUE' }
VERSION : 0.1
   VAR_INPUT
      Pri_1 : SInt;   // Ưu tiên 1
      Pri_2 : SInt;   // Ưu tiên 2
      Pri_3 : SInt;   // Ưu tiên 3
      Pri_4 : SInt;   // Ưu tiên 4
      Pri_5 : SInt;   // Ưu tiên 5
      Pri_6 : SInt;   // Ưu tiên 6
      Pri_7 : SInt;   // Ưu tiên 7
      Pri_8 : SInt;   // Ưu tiên 8
      Pri_9 : SInt;   // Ưu tiên 9
      Pri_10 : SInt;   // Ưu tiên 10
      Pri_11 : SInt;   // Ưu tiên 11
      Pri_12 : SInt;   // Ưu tiên 12
   END_VAR
   VAR_OUTPUT
      Up_Called_F2 : Bool;
      Up_Called_F3 : Bool;
      Up_Called_F4 : Bool;
      Up_Called_F5 : Bool;
      Up_Called_F6 : Bool;
      Down_Called_F1 : Bool;
      Down_Called_F2 : Bool;
      Down_Called_F3 : Bool;
      Down_Called_F4 : Bool;
      Down_Called_F5 : Bool;
   END_VAR
BEGIN
   // KIỂM TRA CÓ GỌI THANG HAY KHÔNG
   // TẦNG 1
   IF #Pri_1 = 11 THEN
       #Down_Called_F1 := 1;
   ELSIF #Pri_2 = 11 THEN
       #Down_Called_F1 := 1;
   ELSIF #Pri_3 = 11 THEN
       #Down_Called_F1 := 1;
   ELSIF #Pri_4 = 11 THEN
       #Down_Called_F1 := 1;
   ELSIF #Pri_5 = 11 THEN
       #Down_Called_F1 := 1;
   ELSIF #Pri_6 = 11 THEN
       #Down_Called_F1 := 1;
   ELSIF #Pri_7 = 11 THEN
       #Down_Called_F1 := 1;
   ELSIF #Pri_8 = 11 THEN
       #Down_Called_F1 := 1;

   ELSE
       #Down_Called_F1 := 0;
       ;
   END_IF;

   // TẦNG 2
   // HẠ
   IF #Pri_1 = 20 THEN
       #Down_Called_F2 := 1;
   ELSIF #Pri_2 = 20 THEN
       #Down_Called_F2 := 1;
   ELSIF #Pri_3 = 20 THEN
       #Down_Called_F2 := 1;
   ELSIF #Pri_4 = 20 THEN
       #Down_Called_F2 := 1;
   ELSIF #Pri_5 = 20 THEN
       #Down_Called_F2 := 1;
   ELSIF #Pri_6 = 20 THEN
       #Down_Called_F2 := 1;
   ELSIF #Pri_7 = 20 THEN
       #Down_Called_F2 := 1;
   ELSIF #Pri_8 = 20 THEN
       #Down_Called_F2 := 1;

   ELSE
       #Down_Called_F2 := 0;
       ;
   END_IF;
   // NÂNG
   IF #Pri_1 = 21 THEN
       #Up_Called_F2 := 1;
   ELSIF #Pri_2 = 21 THEN
       #Up_Called_F2 := 1;
   ELSIF #Pri_3 = 21 THEN
       #Up_Called_F2 := 1;
   ELSIF #Pri_4 = 21 THEN
       #Up_Called_F2 := 1;
   ELSIF #Pri_5 = 21 THEN
       #Up_Called_F2 := 1;
   ELSIF #Pri_6 = 21 THEN
       #Up_Called_F2 := 1;
   ELSIF #Pri_7 = 21 THEN
       #Up_Called_F2 := 1;
   ELSIF #Pri_8 = 21 THEN
       #Up_Called_F2 := 1;

   ELSE
       #Up_Called_F2 := 0;
       ;
   END_IF;
   // TẦNG 3
   // HẠ
   IF #Pri_1 = 30 THEN
       #Down_Called_F3 := 1;
   ELSIF #Pri_2 = 30 THEN
       #Down_Called_F3 := 1;
   ELSIF #Pri_3 = 30 THEN
       #Down_Called_F3 := 1;
   ELSIF #Pri_4 = 30 THEN
       #Down_Called_F3 := 1;
   ELSIF #Pri_5 = 30 THEN
       #Down_Called_F3 := 1;
   ELSIF #Pri_6 = 30 THEN
       #Down_Called_F3 := 1;
   ELSIF #Pri_7 = 30 THEN
       #Down_Called_F3 := 1;
   ELSIF #Pri_8 = 30 THEN
       #Down_Called_F3 := 1;

   ELSE
       #Down_Called_F3 := 0;
       ;
   END_IF;
   // NÂNG
   IF #Pri_1 = 31 THEN
       #Up_Called_F3 := 1;
   ELSIF #Pri_2 = 31 THEN
       #Up_Called_F3 := 1;
   ELSIF #Pri_3 = 31 THEN
       #Up_Called_F3 := 1;
   ELSIF #Pri_4 = 31 THEN
       #Up_Called_F3 := 1;
   ELSIF #Pri_5 = 31 THEN
       #Up_Called_F3 := 1;
   ELSIF #Pri_6 = 31 THEN
       #Up_Called_F3 := 1;
   ELSIF #Pri_7 = 31 THEN
       #Up_Called_F3 := 1;
   ELSIF #Pri_8 = 31 THEN
       #Up_Called_F3 := 1;

   ELSE
       #Up_Called_F3 := 0;
       ;
   END_IF;
   // TẦNG 4
   // HẠ
   IF #Pri_1 = 40 THEN
       #Down_Called_F4 := 1;
   ELSIF #Pri_2 = 40 THEN
       #Down_Called_F4 := 1;
   ELSIF #Pri_3 = 40 THEN
       #Down_Called_F4 := 1;
   ELSIF #Pri_4 = 40 THEN
       #Down_Called_F4 := 1;
   ELSIF #Pri_5 = 40 THEN
       #Down_Called_F4 := 1;
   ELSIF #Pri_6 = 40 THEN
       #Down_Called_F4 := 1;
   ELSIF #Pri_7 = 40 THEN
       #Down_Called_F4 := 1;
   ELSIF #Pri_8 = 40 THEN
       #Down_Called_F4 := 1;

   ELSE
       #Down_Called_F4 := 0;
       ;
   END_IF;
END_FUNCTION

FUNCTION "7.FC_DOOR_CONTROL" : Void   // FC7, LAD
{ S7_Optimized_Access := 'TRUE' }
VERSION : 0.1
   VAR_INPUT
      Ext_Door_Open_Rq : Bool;   // Yêu cầu mở cửa từ FC12
      Setting_Open_Delay_Time : Time;   // Thời gian mở cửa
      Setting_Extreme_Time : Time;   // Đặt thời gian giới hạn khi có lệnh gọi mà cửa không làm gì
   END_VAR
   VAR_OUTPUT
      Pulse_Door_Lock : Bool;
      Door_Open : Bool;
      Door_Close : Bool;
      Alarm_Weight : Bool;
   END_VAR
   VAR_TEMP
      Temp_OP_Delay_Time : Time;
      Temp_Extreme_Time : Time;
   END_VAR
   VAR_TEMP   // added for the SCL form of the ladder/FBD networks
      _w1 : Bool;
      _w2 : Bool;
   END_VAR
BEGIN

REGION Network 1: SETTING TIME (X100) VÌ CÀI ĐẶT LÀ MILI GIÂY (BECAUSE SETTING IS MILISECON)
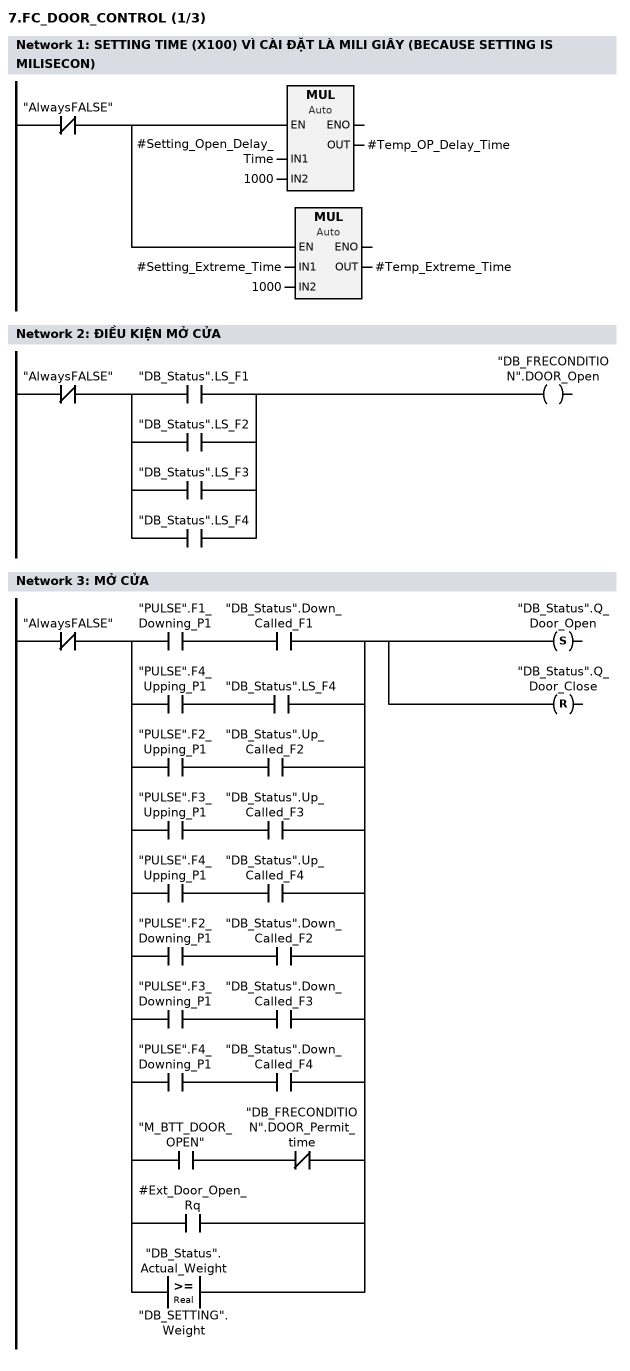
   RUNG wire#powerrail
      I_Contact( "AlwaysFALSE" )
      wire#w1
      Mul(in1 := #Setting_Open_Delay_Time, in2 := 1000, out => #Temp_OP_Delay_Time)
   END_RUNG
   RUNG wire#w1
      Mul(in1 := #Setting_Extreme_Time, in2 := 1000, out => #Temp_Extreme_Time)
   END_RUNG
   // the same network as SCL:
   IF NOT "AlwaysFALSE" THEN
       #Temp_OP_Delay_Time := #Setting_Open_Delay_Time * 1000;
       #Temp_Extreme_Time := #Setting_Extreme_Time * 1000;
   END_IF;
END_REGION

REGION Network 2: ĐIỀU KIỆN MỞ CỬA
   RUNG wire#powerrail
      I_Contact( "AlwaysFALSE" )
      wire#w1
      Contact( "DB_Status".LS_F1 )
      wire#w2
      Coil( "DB_FRECONDITION".DOOR_Open )
   END_RUNG
   RUNG wire#w1
      Contact( "DB_Status".LS_F2 )
   END_RUNG wire#w2
   RUNG wire#w1
      Contact( "DB_Status".LS_F3 )
   END_RUNG wire#w2
   RUNG wire#w1
      Contact( "DB_Status".LS_F4 )
   END_RUNG wire#w2
   // the same network as SCL:
   "DB_FRECONDITION".DOOR_Open := NOT "AlwaysFALSE" AND ("DB_Status".LS_F1 OR "DB_Status".LS_F2 OR "DB_Status".LS_F3 OR "DB_Status".LS_F4);
END_REGION

REGION Network 3: MỞ CỬA
   RUNG wire#powerrail
      I_Contact( "AlwaysFALSE" )
      wire#w1
      Contact( "PULSE".F1_Downing_P1 )
      Contact( "DB_Status".Down_Called_F1 )
      wire#w2
      S_Coil( "DB_Status".Q_Door_Open )
   END_RUNG
   RUNG wire#w1
      Contact( "PULSE".F4_Upping_P1 )
      Contact( "DB_Status".LS_F4 )
   END_RUNG wire#w2
   RUNG wire#w1
      Contact( "PULSE".F2_Upping_P1 )
      Contact( "DB_Status".Up_Called_F2 )
   END_RUNG wire#w2
   RUNG wire#w1
      Contact( "PULSE".F3_Upping_P1 )
      Contact( "DB_Status".Up_Called_F3 )
   END_RUNG wire#w2
   RUNG wire#w1
      Contact( "PULSE".F4_Upping_P1 )
      Contact( "DB_Status".Up_Called_F4 )
   END_RUNG wire#w2
   RUNG wire#w1
      Contact( "PULSE".F2_Downing_P1 )
      Contact( "DB_Status".Down_Called_F2 )
   END_RUNG wire#w2
   RUNG wire#w1
      Contact( "PULSE".F3_Downing_P1 )
      Contact( "DB_Status".Down_Called_F3 )
   END_RUNG wire#w2
   RUNG wire#w1
      Contact( "PULSE".F4_Downing_P1 )
      Contact( "DB_Status".Down_Called_F4 )
   END_RUNG wire#w2
   RUNG wire#w1
      Contact( "M_BTT_DOOR_OPEN" )
      I_Contact( "DB_FRECONDITION".DOOR_Permit_time )
   END_RUNG wire#w2
   RUNG wire#w1
      Contact( #Ext_Door_Open_Rq )
   END_RUNG wire#w2
   RUNG wire#w1
      { S7_Templates := "SrcType := Real" } GE_Contact(in1 := "DB_Status".Actual_Weight, in2 := "DB_SETTING".Weight)
   END_RUNG wire#w2
   RUNG wire#w2
      R_Coil( "DB_Status".Q_Door_Close )
   END_RUNG
   // the same network as SCL:
   IF NOT "AlwaysFALSE" AND (("PULSE".F1_Downing_P1 AND "DB_Status".Down_Called_F1) OR ("PULSE".F4_Upping_P1 AND "DB_Status".LS_F4) OR ("PULSE".F2_Upping_P1 AND "DB_Status".Up_Called_F2) OR ("PULSE".F3_Upping_P1 AND "DB_Status".Up_Called_F3) OR ("PULSE".F4_Upping_P1 AND "DB_Status".Up_Called_F4) OR ("PULSE".F2_Downing_P1 AND "DB_Status".Down_Called_F2) OR ("PULSE".F3_Downing_P1 AND "DB_Status".Down_Called_F3) OR ("PULSE".F4_Downing_P1 AND "DB_Status".Down_Called_F4) OR ("M_BTT_DOOR_OPEN" AND NOT "DB_FRECONDITION".DOOR_Permit_time) OR #Ext_Door_Open_Rq OR ("DB_Status".Actual_Weight >= "DB_SETTING".Weight)) THEN
       "DB_Status".Q_Door_Open := TRUE;
       "DB_Status".Q_Door_Close := FALSE;
   END_IF;
END_REGION

REGION Network 4: DELAY MỞ CỬA
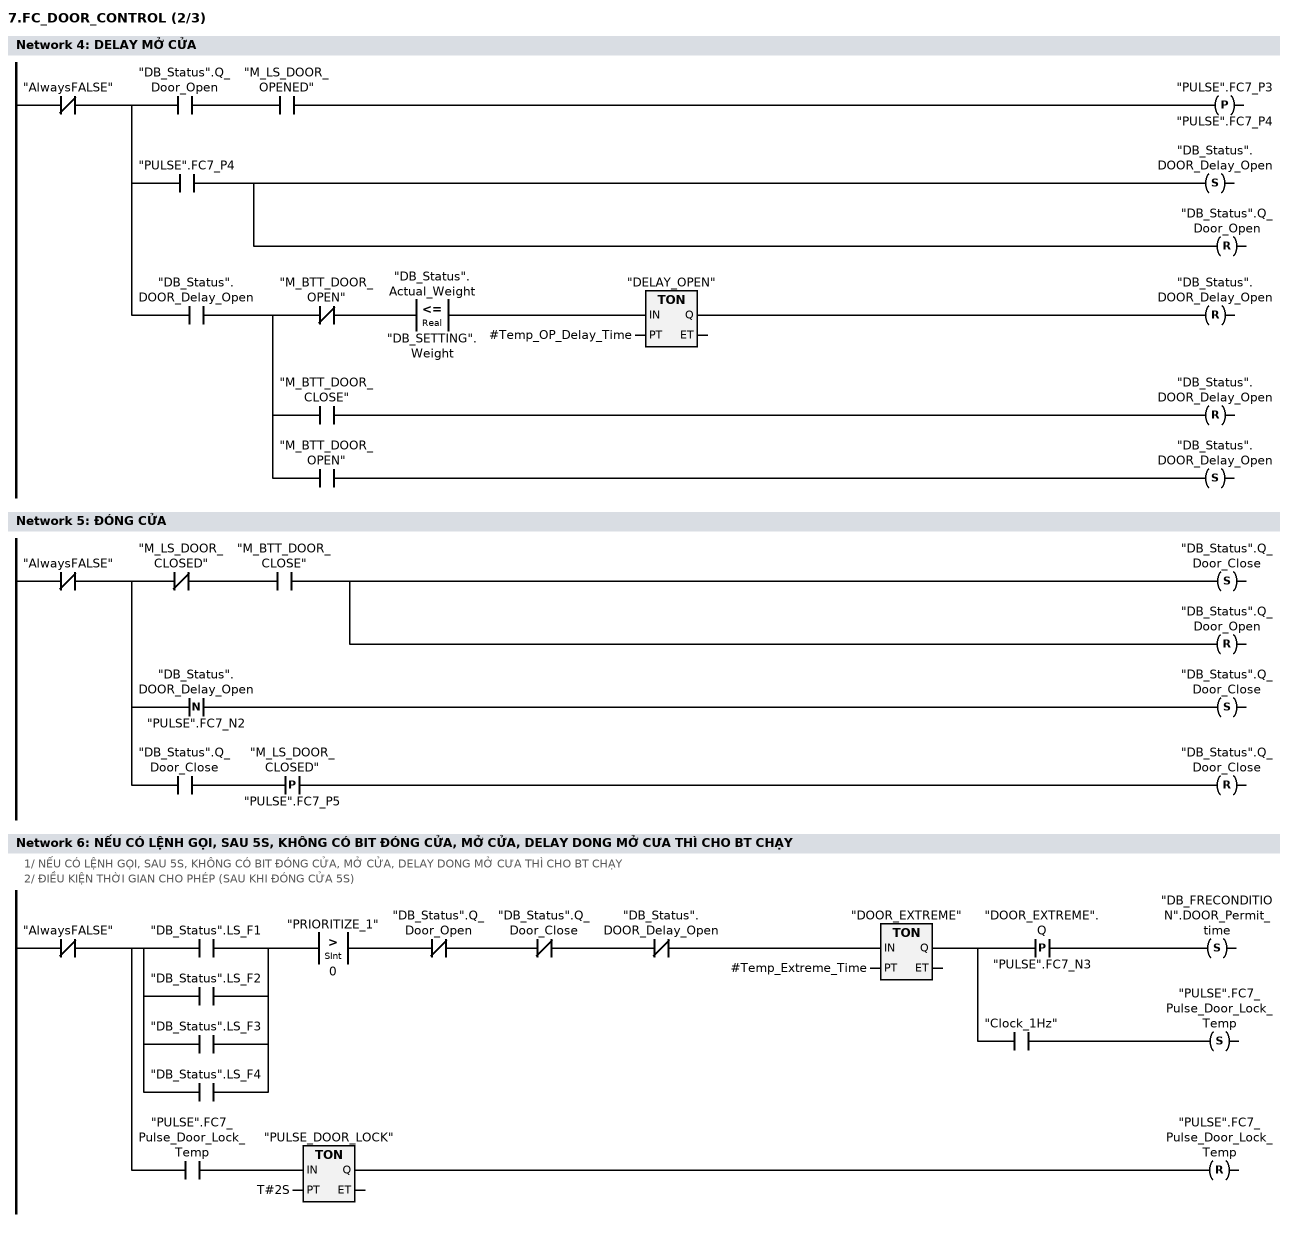
   #_w1 := NOT "AlwaysFALSE" AND "DB_Status".Q_Door_Open AND "M_LS_DOOR_OPENED";
   "PULSE".FC7_P3 := #_w1 AND NOT "PULSE".FC7_P4;   // rising edge
   "PULSE".FC7_P4 := #_w1;
   IF NOT "AlwaysFALSE" AND "PULSE".FC7_P4 THEN
       "DB_Status".DOOR_Delay_Open := TRUE;
       "DB_Status".Q_Door_Open := FALSE;
   END_IF;
   #_w2 := NOT "AlwaysFALSE" AND "DB_Status".DOOR_Delay_Open;
   "DELAY_OPEN".TON(IN := #_w2 AND NOT "M_BTT_DOOR_OPEN" AND ("DB_Status".Actual_Weight <= "DB_SETTING".Weight),
                    PT := #Temp_OP_Delay_Time);
   IF "DELAY_OPEN".Q THEN "DB_Status".DOOR_Delay_Open := FALSE; END_IF;
   IF #_w2 AND "M_BTT_DOOR_CLOSE" THEN "DB_Status".DOOR_Delay_Open := FALSE; END_IF;
   IF #_w2 AND "M_BTT_DOOR_OPEN" THEN "DB_Status".DOOR_Delay_Open := TRUE; END_IF;
END_REGION

REGION Network 5: ĐÓNG CỬA
   RUNG wire#powerrail
      I_Contact( "AlwaysFALSE" )
      wire#w1
      I_Contact( "M_LS_DOOR_CLOSED" )
      Contact( "M_BTT_DOOR_CLOSE" )
      wire#w2
      S_Coil( "DB_Status".Q_Door_Close )
   END_RUNG
   RUNG wire#w2
      R_Coil( "DB_Status".Q_Door_Open )
   END_RUNG
   RUNG wire#w1
      N_Contact(operand := "DB_Status".DOOR_Delay_Open, bit := "PULSE".FC7_N2)
      S_Coil( "DB_Status".Q_Door_Close )
   END_RUNG
   RUNG wire#w1
      Contact( "DB_Status".Q_Door_Close )
      P_Contact(operand := "M_LS_DOOR_CLOSED", bit := "PULSE".FC7_P5)
      R_Coil( "DB_Status".Q_Door_Close )
   END_RUNG
   // the same network as SCL:
   IF NOT "AlwaysFALSE" AND NOT "M_LS_DOOR_CLOSED" AND "M_BTT_DOOR_CLOSE" THEN
       "DB_Status".Q_Door_Close := TRUE;
       "DB_Status".Q_Door_Open := FALSE;
   END_IF;
   #_w1 := NOT "AlwaysFALSE" AND NOT "DB_Status".DOOR_Delay_Open AND "PULSE".FC7_N2;   // falling edge of "DB_Status".DOOR_Delay_Open
   "PULSE".FC7_N2 := "DB_Status".DOOR_Delay_Open;
   IF #_w1 THEN "DB_Status".Q_Door_Close := TRUE; END_IF;
   #_w2 := NOT "AlwaysFALSE" AND "DB_Status".Q_Door_Close AND "M_LS_DOOR_CLOSED" AND NOT "PULSE".FC7_P5;   // rising edge of "M_LS_DOOR_CLOSED"
   "PULSE".FC7_P5 := "M_LS_DOOR_CLOSED";
   IF #_w2 THEN "DB_Status".Q_Door_Close := FALSE; END_IF;
END_REGION

REGION Network 6: NẾU CÓ LỆNH GỌI, SAU 5S, KHÔNG CÓ BIT ĐÓNG CỬA, MỞ CỬA, DELAY DONG MỞ CƯA THÌ CHO BT CHẠY
   // 1/ NẾU CÓ LỆNH GỌI, SAU 5S, KHÔNG CÓ BIT ĐÓNG CỬA, MỞ CỬA, DELAY DONG MỞ CƯA THÌ CHO BT CHẠY
   // 2/ ĐIỀU KIỆN THỜI GIAN CHO PHÉP (SAU KHI ĐÓNG CỬA 5S)
   "DOOR_EXTREME".TON(IN := NOT "AlwaysFALSE" AND ("DB_Status".LS_F1 OR "DB_Status".LS_F2 OR "DB_Status".LS_F3 OR "DB_Status".LS_F4) AND ("PRIORITIZE_1" > 0) AND NOT "DB_Status".Q_Door_Open AND NOT "DB_Status".Q_Door_Close AND NOT "DB_Status".DOOR_Delay_Open,
                      PT := #Temp_Extreme_Time);
   #_w1 := "DOOR_EXTREME".Q AND "DOOR_EXTREME".Q AND NOT "PULSE".FC7_N3;   // rising edge of "DOOR_EXTREME".Q
   "PULSE".FC7_N3 := "DOOR_EXTREME".Q;
   IF #_w1 THEN "DB_FRECONDITION".DOOR_Permit_time := TRUE; END_IF;
   IF "DOOR_EXTREME".Q AND "Clock_1Hz" THEN "PULSE".FC7_Pulse_Door_Lock_Temp := TRUE; END_IF;
   "PULSE_DOOR_LOCK".TON(IN := NOT "AlwaysFALSE" AND "PULSE".FC7_Pulse_Door_Lock_Temp, PT := T#2S);
   IF "PULSE_DOOR_LOCK".Q THEN "PULSE".FC7_Pulse_Door_Lock_Temp := FALSE; END_IF;
END_REGION

REGION Network 7: RESET BIT PERMIT
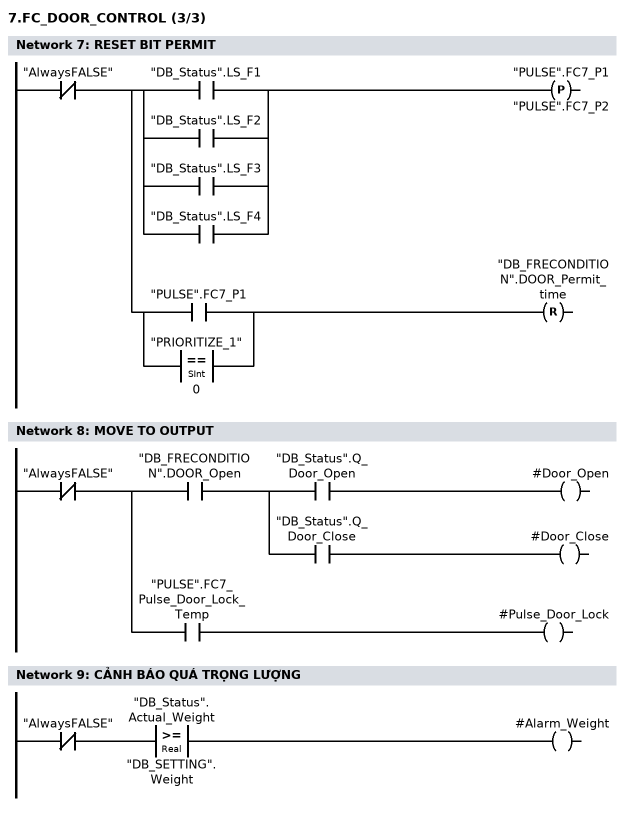
   #_w1 := NOT "AlwaysFALSE" AND ("DB_Status".LS_F1 OR "DB_Status".LS_F2 OR "DB_Status".LS_F3 OR "DB_Status".LS_F4);
   "PULSE".FC7_P1 := #_w1 AND NOT "PULSE".FC7_P2;   // rising edge
   "PULSE".FC7_P2 := #_w1;
   IF NOT "AlwaysFALSE" AND ("PULSE".FC7_P1 OR ("PRIORITIZE_1" = 0)) THEN
       "DB_FRECONDITION".DOOR_Permit_time := FALSE;
   END_IF;
END_REGION

REGION Network 8: MOVE TO OUTPUT
   RUNG wire#powerrail
      I_Contact( "AlwaysFALSE" )
      wire#w1
      Contact( "DB_FRECONDITION".DOOR_Open )
      wire#w2
      Contact( "DB_Status".Q_Door_Open )
      Coil( #Door_Open )
   END_RUNG
   RUNG wire#w2
      Contact( "DB_Status".Q_Door_Close )
      Coil( #Door_Close )
   END_RUNG
   RUNG wire#w1
      Contact( "PULSE".FC7_Pulse_Door_Lock_Temp )
      Coil( #Pulse_Door_Lock )
   END_RUNG
   // the same network as SCL:
   #_w1 := NOT "AlwaysFALSE" AND "DB_FRECONDITION".DOOR_Open;
   #Door_Open := #_w1 AND "DB_Status".Q_Door_Open;
   #Door_Close := #_w1 AND "DB_Status".Q_Door_Close;
   #Pulse_Door_Lock := NOT "AlwaysFALSE" AND "PULSE".FC7_Pulse_Door_Lock_Temp;
END_REGION

REGION Network 9: CẢNH BÁO QUÁ TRỌNG LƯỢNG
   RUNG wire#powerrail
      I_Contact( "AlwaysFALSE" )
      { S7_Templates := "SrcType := Real" } GE_Contact(in1 := "DB_Status".Actual_Weight, in2 := "DB_SETTING".Weight)
      Coil( #Alarm_Weight )
   END_RUNG
   // the same network as SCL:
   #Alarm_Weight := NOT "AlwaysFALSE" AND ("DB_Status".Actual_Weight >= "DB_SETTING".Weight);
END_REGION
END_FUNCTION

FUNCTION "8.FC_SIMULATION" : Void   // FC8, LAD
{ S7_Optimized_Access := 'TRUE' }
VERSION : 0.1
   VAR_TEMP   // added for the SCL form of the ladder/FBD networks
      _w1 : Bool;
      _w2 : Bool;
      _w3 : Bool;
      _w4 : Bool;
   END_VAR
BEGIN

REGION Network 1: MÔ PHỎNG VỊ TRÍ THANG MÁY
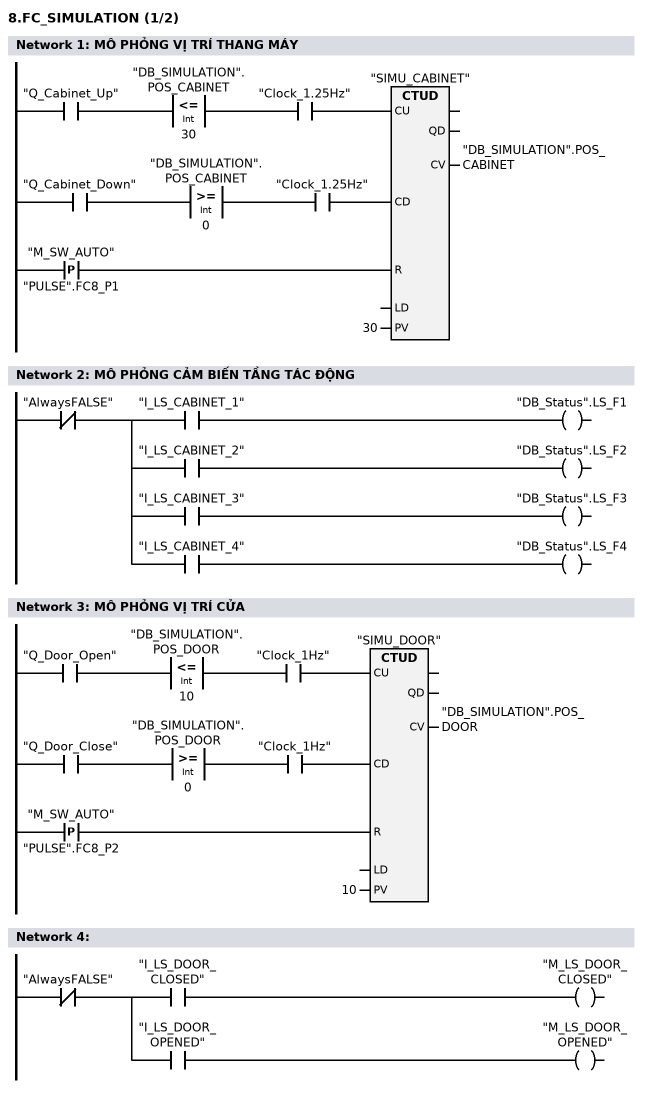
   #_w1 := "M_SW_AUTO" AND NOT "PULSE".FC8_P1;   // rising edge of "M_SW_AUTO"
   "PULSE".FC8_P1 := "M_SW_AUTO";
   "SIMU_CABINET".CTUD(CU := "Q_Cabinet_Up" AND ("DB_SIMULATION".POS_CABINET <= 30) AND "Clock_1.25Hz",
                       CD := "Q_Cabinet_Down" AND ("DB_SIMULATION".POS_CABINET >= 0) AND "Clock_1.25Hz",
                       R := #_w1,
                       PV := 30,
                       CV => "DB_SIMULATION".POS_CABINET);
END_REGION

REGION Network 2: MÔ PHỎNG CẢM BIẾN TẦNG TÁC ĐỘNG
   RUNG wire#powerrail
      I_Contact( "AlwaysFALSE" )
      wire#w1
      Contact( "I_LS_CABINET_1" )
      Coil( "DB_Status".LS_F1 )
   END_RUNG
   RUNG wire#w1
      Contact( "I_LS_CABINET_2" )
      Coil( "DB_Status".LS_F2 )
   END_RUNG
   RUNG wire#w1
      Contact( "I_LS_CABINET_3" )
      Coil( "DB_Status".LS_F3 )
   END_RUNG
   RUNG wire#w1
      Contact( "I_LS_CABINET_4" )
      Coil( "DB_Status".LS_F4 )
   END_RUNG
   // the same network as SCL:
   "DB_Status".LS_F1 := NOT "AlwaysFALSE" AND "I_LS_CABINET_1";
   "DB_Status".LS_F2 := NOT "AlwaysFALSE" AND "I_LS_CABINET_2";
   "DB_Status".LS_F3 := NOT "AlwaysFALSE" AND "I_LS_CABINET_3";
   "DB_Status".LS_F4 := NOT "AlwaysFALSE" AND "I_LS_CABINET_4";
END_REGION

REGION Network 3: MÔ PHỎNG VỊ TRÍ CỬA
   #_w1 := "M_SW_AUTO" AND NOT "PULSE".FC8_P2;   // rising edge of "M_SW_AUTO"
   "PULSE".FC8_P2 := "M_SW_AUTO";
   "SIMU_DOOR".CTUD(CU := "Q_Door_Open" AND ("DB_SIMULATION".POS_DOOR <= 10) AND "Clock_1Hz",
                    CD := "Q_Door_Close" AND ("DB_SIMULATION".POS_DOOR >= 0) AND "Clock_1Hz",
                    R := #_w1,
                    PV := 10,
                    CV => "DB_SIMULATION".POS_DOOR);
END_REGION

REGION Network 4
   RUNG wire#powerrail
      I_Contact( "AlwaysFALSE" )
      wire#w1
      Contact( "I_LS_DOOR_CLOSED" )
      Coil( "M_LS_DOOR_CLOSED" )
   END_RUNG
   RUNG wire#w1
      Contact( "I_LS_DOOR_OPENED" )
      Coil( "M_LS_DOOR_OPENED" )
   END_RUNG
   // the same network as SCL:
   "M_LS_DOOR_CLOSED" := NOT "AlwaysFALSE" AND "I_LS_DOOR_CLOSED";
   "M_LS_DOOR_OPENED" := NOT "AlwaysFALSE" AND "I_LS_DOOR_OPENED";
END_REGION

REGION Network 5: HIỂN THỊ VỊ TRÍ CỬA (DISPLAY DOOR POSITION IN WINCC)
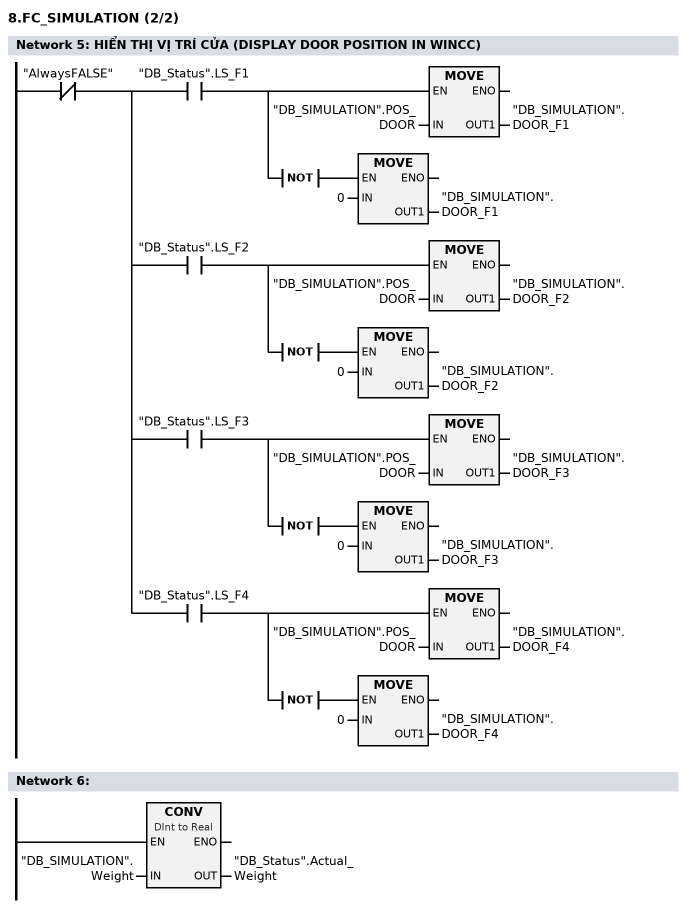
   RUNG wire#powerrail
      I_Contact( "AlwaysFALSE" )
      wire#w1
      Contact( "DB_Status".LS_F1 )
      wire#w2
      Move(in := "DB_SIMULATION".POS_DOOR, out1 => "DB_SIMULATION".DOOR_F1)
   END_RUNG
   RUNG wire#w2
      Not()
      Move(in := 0, out1 => "DB_SIMULATION".DOOR_F1)
   END_RUNG
   RUNG wire#w1
      Contact( "DB_Status".LS_F2 )
      wire#w3
      Move(in := "DB_SIMULATION".POS_DOOR, out1 => "DB_SIMULATION".DOOR_F2)
   END_RUNG
   RUNG wire#w3
      Not()
      Move(in := 0, out1 => "DB_SIMULATION".DOOR_F2)
   END_RUNG
   RUNG wire#w1
      Contact( "DB_Status".LS_F3 )
      wire#w4
      Move(in := "DB_SIMULATION".POS_DOOR, out1 => "DB_SIMULATION".DOOR_F3)
   END_RUNG
   RUNG wire#w4
      Not()
      Move(in := 0, out1 => "DB_SIMULATION".DOOR_F3)
   END_RUNG
   RUNG wire#w1
      Contact( "DB_Status".LS_F4 )
      wire#w5
      Move(in := "DB_SIMULATION".POS_DOOR, out1 => "DB_SIMULATION".DOOR_F4)
   END_RUNG
   RUNG wire#w5
      Not()
      Move(in := 0, out1 => "DB_SIMULATION".DOOR_F4)
   END_RUNG
   // the same network as SCL:
   #_w1 := NOT "AlwaysFALSE" AND "DB_Status".LS_F1;
   IF #_w1 THEN "DB_SIMULATION".DOOR_F1 := "DB_SIMULATION".POS_DOOR; END_IF;
   IF NOT #_w1 THEN "DB_SIMULATION".DOOR_F1 := 0; END_IF;
   #_w2 := NOT "AlwaysFALSE" AND "DB_Status".LS_F2;
   IF #_w2 THEN "DB_SIMULATION".DOOR_F2 := "DB_SIMULATION".POS_DOOR; END_IF;
   IF NOT #_w2 THEN "DB_SIMULATION".DOOR_F2 := 0; END_IF;
   #_w3 := NOT "AlwaysFALSE" AND "DB_Status".LS_F3;
   IF #_w3 THEN "DB_SIMULATION".DOOR_F3 := "DB_SIMULATION".POS_DOOR; END_IF;
   IF NOT #_w3 THEN "DB_SIMULATION".DOOR_F3 := 0; END_IF;
   #_w4 := NOT "AlwaysFALSE" AND "DB_Status".LS_F4;
   IF #_w4 THEN "DB_SIMULATION".DOOR_F4 := "DB_SIMULATION".POS_DOOR; END_IF;
   IF NOT #_w4 THEN "DB_SIMULATION".DOOR_F4 := 0; END_IF;
END_REGION

REGION Network 6
   RUNG wire#powerrail
      { S7_Templates := "[SrcType := DInt, DestType := Real]" } Convert(in := "DB_SIMULATION".Weight, out => "DB_Status".Actual_Weight)
   END_RUNG
   // the same network as SCL:
   "DB_Status".Actual_Weight := DINT_TO_REAL("DB_SIMULATION".Weight);
END_REGION
END_FUNCTION

FUNCTION "Moving" : Void   // FC9, LAD
{ S7_Optimized_Access := 'TRUE' }
VERSION : 0.1
BEGIN

REGION Network 1
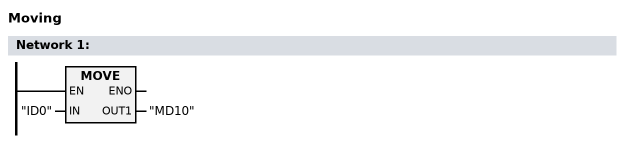
   RUNG wire#powerrail
      Move(in := "ID0", out1 => "MD10")
   END_RUNG
   // the same network as SCL:
   "MD10" := "ID0";
END_REGION
END_FUNCTION

FUNCTION "10.FC_BUTTON_CONTROL" : Void   // FC10, LAD
{ S7_Optimized_Access := 'TRUE' }
VERSION : 0.1
BEGIN

REGION Network 1: LỰA CHỌN TẦNG 1
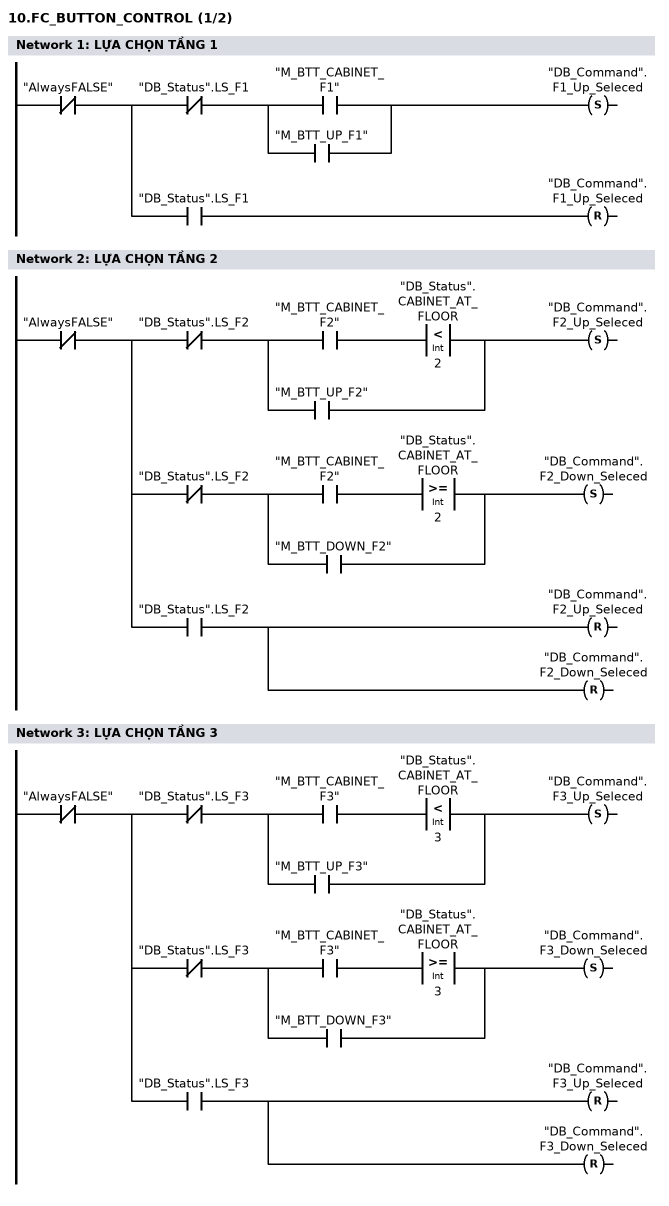
   RUNG wire#powerrail
      I_Contact( "AlwaysFALSE" )
      wire#w1
      I_Contact( "DB_Status".LS_F1 )
      wire#w2
      Contact( "M_BTT_CABINET_F1" )
      wire#w3
      S_Coil( "DB_Command".F1_Up_Seleced )
   END_RUNG
   RUNG wire#w2
      Contact( "M_BTT_UP_F1" )
   END_RUNG wire#w3
   RUNG wire#w1
      Contact( "DB_Status".LS_F1 )
      R_Coil( "DB_Command".F1_Up_Seleced )
   END_RUNG
   // the same network as SCL:
   IF NOT "AlwaysFALSE" AND NOT "DB_Status".LS_F1 AND ("M_BTT_CABINET_F1" OR "M_BTT_UP_F1") THEN
       "DB_Command".F1_Up_Seleced := TRUE;
   END_IF;
   IF NOT "AlwaysFALSE" AND "DB_Status".LS_F1 THEN "DB_Command".F1_Up_Seleced := FALSE; END_IF;
END_REGION

REGION Network 2: LỰA CHỌN TẦNG 2
   RUNG wire#powerrail
      I_Contact( "AlwaysFALSE" )
      wire#w1
      I_Contact( "DB_Status".LS_F2 )
      wire#w2
      Contact( "M_BTT_CABINET_F2" )
      { S7_Templates := "SrcType := Int" } LT_Contact(in1 := "DB_Status".CABINET_AT_FLOOR, in2 := 2)
      wire#w3
      S_Coil( "DB_Command".F2_Up_Seleced )
   END_RUNG
   RUNG wire#w2
      Contact( "M_BTT_UP_F2" )
   END_RUNG wire#w3
   RUNG wire#w1
      I_Contact( "DB_Status".LS_F2 )
      wire#w4
      Contact( "M_BTT_CABINET_F2" )
      { S7_Templates := "SrcType := Int" } GE_Contact(in1 := "DB_Status".CABINET_AT_FLOOR, in2 := 2)
      wire#w5
      S_Coil( "DB_Command".F2_Down_Seleced )
   END_RUNG
   RUNG wire#w4
      Contact( "M_BTT_DOWN_F2" )
   END_RUNG wire#w5
   RUNG wire#w1
      Contact( "DB_Status".LS_F2 )
      wire#w6
      R_Coil( "DB_Command".F2_Up_Seleced )
   END_RUNG
   RUNG wire#w6
      R_Coil( "DB_Command".F2_Down_Seleced )
   END_RUNG
   // the same network as SCL:
   IF NOT "AlwaysFALSE" AND NOT "DB_Status".LS_F2 AND (("M_BTT_CABINET_F2" AND ("DB_Status".CABINET_AT_FLOOR < 2)) OR "M_BTT_UP_F2") THEN
       "DB_Command".F2_Up_Seleced := TRUE;
   END_IF;
   IF NOT "AlwaysFALSE" AND NOT "DB_Status".LS_F2 AND (("M_BTT_CABINET_F2" AND ("DB_Status".CABINET_AT_FLOOR >= 2)) OR "M_BTT_DOWN_F2") THEN
       "DB_Command".F2_Down_Seleced := TRUE;
   END_IF;
   IF NOT "AlwaysFALSE" AND "DB_Status".LS_F2 THEN
       "DB_Command".F2_Up_Seleced := FALSE;
       "DB_Command".F2_Down_Seleced := FALSE;
   END_IF;
END_REGION

REGION Network 3: LỰA CHỌN TẦNG 3
   RUNG wire#powerrail
      I_Contact( "AlwaysFALSE" )
      wire#w1
      I_Contact( "DB_Status".LS_F3 )
      wire#w2
      Contact( "M_BTT_CABINET_F3" )
      { S7_Templates := "SrcType := Int" } LT_Contact(in1 := "DB_Status".CABINET_AT_FLOOR, in2 := 3)
      wire#w3
      S_Coil( "DB_Command".F3_Up_Seleced )
   END_RUNG
   RUNG wire#w2
      Contact( "M_BTT_UP_F3" )
   END_RUNG wire#w3
   RUNG wire#w1
      I_Contact( "DB_Status".LS_F3 )
      wire#w4
      Contact( "M_BTT_CABINET_F3" )
      { S7_Templates := "SrcType := Int" } GE_Contact(in1 := "DB_Status".CABINET_AT_FLOOR, in2 := 3)
      wire#w5
      S_Coil( "DB_Command".F3_Down_Seleced )
   END_RUNG
   RUNG wire#w4
      Contact( "M_BTT_DOWN_F3" )
   END_RUNG wire#w5
   RUNG wire#w1
      Contact( "DB_Status".LS_F3 )
      wire#w6
      R_Coil( "DB_Command".F3_Up_Seleced )
   END_RUNG
   RUNG wire#w6
      R_Coil( "DB_Command".F3_Down_Seleced )
   END_RUNG
   // the same network as SCL:
   IF NOT "AlwaysFALSE" AND NOT "DB_Status".LS_F3 AND (("M_BTT_CABINET_F3" AND ("DB_Status".CABINET_AT_FLOOR < 3)) OR "M_BTT_UP_F3") THEN
       "DB_Command".F3_Up_Seleced := TRUE;
   END_IF;
   IF NOT "AlwaysFALSE" AND NOT "DB_Status".LS_F3 AND (("M_BTT_CABINET_F3" AND ("DB_Status".CABINET_AT_FLOOR >= 3)) OR "M_BTT_DOWN_F3") THEN
       "DB_Command".F3_Down_Seleced := TRUE;
   END_IF;
   IF NOT "AlwaysFALSE" AND "DB_Status".LS_F3 THEN
       "DB_Command".F3_Up_Seleced := FALSE;
       "DB_Command".F3_Down_Seleced := FALSE;
   END_IF;
END_REGION

REGION Network 4: LỰA CHỌN TẦNG 4
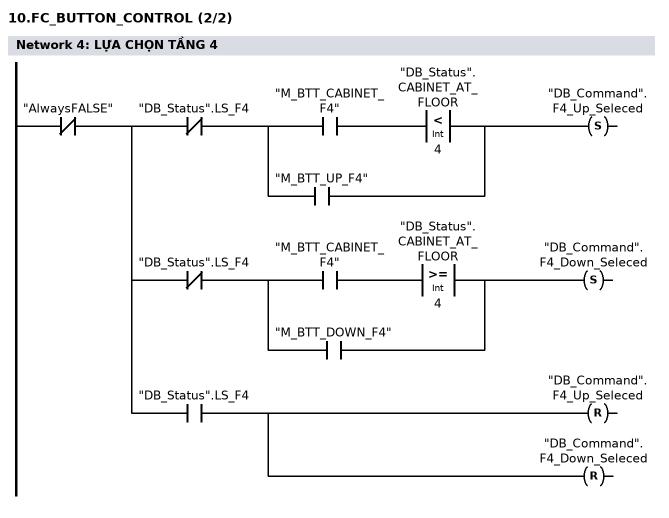
   RUNG wire#powerrail
      I_Contact( "AlwaysFALSE" )
      wire#w1
      I_Contact( "DB_Status".LS_F4 )
      wire#w2
      Contact( "M_BTT_CABINET_F4" )
      { S7_Templates := "SrcType := Int" } LT_Contact(in1 := "DB_Status".CABINET_AT_FLOOR, in2 := 4)
      wire#w3
      S_Coil( "DB_Command".F4_Up_Seleced )
   END_RUNG
   RUNG wire#w2
      Contact( "M_BTT_UP_F4" )
   END_RUNG wire#w3
   RUNG wire#w1
      I_Contact( "DB_Status".LS_F4 )
      wire#w4
      Contact( "M_BTT_CABINET_F4" )
      { S7_Templates := "SrcType := Int" } GE_Contact(in1 := "DB_Status".CABINET_AT_FLOOR, in2 := 4)
      wire#w5
      S_Coil( "DB_Command".F4_Down_Seleced )
   END_RUNG
   RUNG wire#w4
      Contact( "M_BTT_DOWN_F4" )
   END_RUNG wire#w5
   RUNG wire#w1
      Contact( "DB_Status".LS_F4 )
      wire#w6
      R_Coil( "DB_Command".F4_Up_Seleced )
   END_RUNG
   RUNG wire#w6
      R_Coil( "DB_Command".F4_Down_Seleced )
   END_RUNG
   // the same network as SCL:
   IF NOT "AlwaysFALSE" AND NOT "DB_Status".LS_F4 AND (("M_BTT_CABINET_F4" AND ("DB_Status".CABINET_AT_FLOOR < 4)) OR "M_BTT_UP_F4") THEN
       "DB_Command".F4_Up_Seleced := TRUE;
   END_IF;
   IF NOT "AlwaysFALSE" AND NOT "DB_Status".LS_F4 AND (("M_BTT_CABINET_F4" AND ("DB_Status".CABINET_AT_FLOOR >= 4)) OR "M_BTT_DOWN_F4") THEN
       "DB_Command".F4_Down_Seleced := TRUE;
   END_IF;
   IF NOT "AlwaysFALSE" AND "DB_Status".LS_F4 THEN
       "DB_Command".F4_Up_Seleced := FALSE;
       "DB_Command".F4_Down_Seleced := FALSE;
   END_IF;
END_REGION
END_FUNCTION

FUNCTION "11.FC_LAMP_CONTROL" : Void   // FC11, LAD
{ S7_Optimized_Access := 'TRUE' }
VERSION : 0.1
   VAR_TEMP   // added for the SCL form of the ladder/FBD networks
      _w1 : Bool;
   END_VAR
BEGIN

REGION Network 1: ĐÈN ĐIỀU KHIỂN
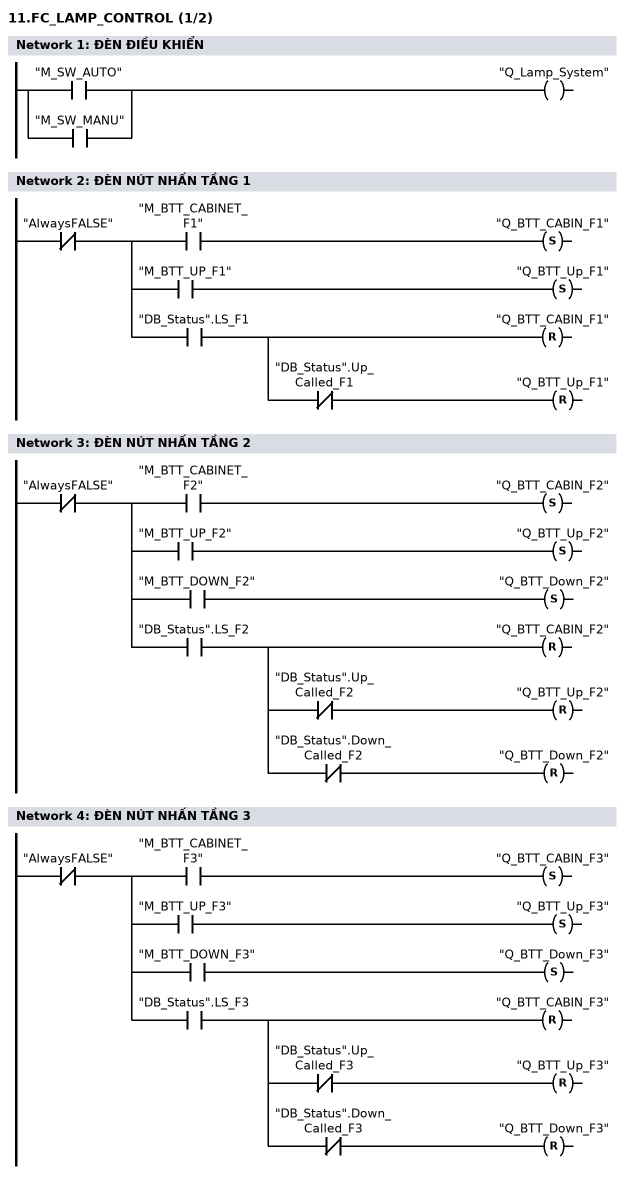
   RUNG wire#powerrail
      Contact( "M_SW_AUTO" )
      wire#w1
      Coil( "Q_Lamp_System" )
   END_RUNG
   RUNG wire#powerrail
      Contact( "M_SW_MANU" )
   END_RUNG wire#w1
   // the same network as SCL:
   "Q_Lamp_System" := "M_SW_AUTO" OR "M_SW_MANU";
END_REGION

REGION Network 2: ĐÈN NÚT NHẤN TẦNG 1
   RUNG wire#powerrail
      I_Contact( "AlwaysFALSE" )
      wire#w1
      Contact( "M_BTT_CABINET_F1" )
      S_Coil( "Q_BTT_CABIN_F1" )
   END_RUNG
   RUNG wire#w1
      Contact( "M_BTT_UP_F1" )
      S_Coil( "Q_BTT_Up_F1" )
   END_RUNG
   RUNG wire#w1
      Contact( "DB_Status".LS_F1 )
      wire#w2
      R_Coil( "Q_BTT_CABIN_F1" )
   END_RUNG
   RUNG wire#w2
      I_Contact( "DB_Status".Up_Called_F1 )
      R_Coil( "Q_BTT_Up_F1" )
   END_RUNG
   // the same network as SCL:
   IF NOT "AlwaysFALSE" AND "M_BTT_CABINET_F1" THEN "Q_BTT_CABIN_F1" := TRUE; END_IF;
   IF NOT "AlwaysFALSE" AND "M_BTT_UP_F1" THEN "Q_BTT_Up_F1" := TRUE; END_IF;
   #_w1 := NOT "AlwaysFALSE" AND "DB_Status".LS_F1;
   IF #_w1 THEN "Q_BTT_CABIN_F1" := FALSE; END_IF;
   IF #_w1 AND NOT "DB_Status".Up_Called_F1 THEN "Q_BTT_Up_F1" := FALSE; END_IF;
END_REGION

REGION Network 3: ĐÈN NÚT NHẤN TẦNG 2
   RUNG wire#powerrail
      I_Contact( "AlwaysFALSE" )
      wire#w1
      Contact( "M_BTT_CABINET_F2" )
      S_Coil( "Q_BTT_CABIN_F2" )
   END_RUNG
   RUNG wire#w1
      Contact( "M_BTT_UP_F2" )
      S_Coil( "Q_BTT_Up_F2" )
   END_RUNG
   RUNG wire#w1
      Contact( "M_BTT_DOWN_F2" )
      S_Coil( "Q_BTT_Down_F2" )
   END_RUNG
   RUNG wire#w1
      Contact( "DB_Status".LS_F2 )
      wire#w2
      R_Coil( "Q_BTT_CABIN_F2" )
   END_RUNG
   RUNG wire#w2
      I_Contact( "DB_Status".Up_Called_F2 )
      R_Coil( "Q_BTT_Up_F2" )
   END_RUNG
   RUNG wire#w2
      I_Contact( "DB_Status".Down_Called_F2 )
      R_Coil( "Q_BTT_Down_F2" )
   END_RUNG
   // the same network as SCL:
   IF NOT "AlwaysFALSE" AND "M_BTT_CABINET_F2" THEN "Q_BTT_CABIN_F2" := TRUE; END_IF;
   IF NOT "AlwaysFALSE" AND "M_BTT_UP_F2" THEN "Q_BTT_Up_F2" := TRUE; END_IF;
   IF NOT "AlwaysFALSE" AND "M_BTT_DOWN_F2" THEN "Q_BTT_Down_F2" := TRUE; END_IF;
   #_w1 := NOT "AlwaysFALSE" AND "DB_Status".LS_F2;
   IF #_w1 THEN "Q_BTT_CABIN_F2" := FALSE; END_IF;
   IF #_w1 AND NOT "DB_Status".Up_Called_F2 THEN "Q_BTT_Up_F2" := FALSE; END_IF;
   IF #_w1 AND NOT "DB_Status".Down_Called_F2 THEN "Q_BTT_Down_F2" := FALSE; END_IF;
END_REGION

REGION Network 4: ĐÈN NÚT NHẤN TẦNG 3
   RUNG wire#powerrail
      I_Contact( "AlwaysFALSE" )
      wire#w1
      Contact( "M_BTT_CABINET_F3" )
      S_Coil( "Q_BTT_CABIN_F3" )
   END_RUNG
   RUNG wire#w1
      Contact( "M_BTT_UP_F3" )
      S_Coil( "Q_BTT_Up_F3" )
   END_RUNG
   RUNG wire#w1
      Contact( "M_BTT_DOWN_F3" )
      S_Coil( "Q_BTT_Down_F3" )
   END_RUNG
   RUNG wire#w1
      Contact( "DB_Status".LS_F3 )
      wire#w2
      R_Coil( "Q_BTT_CABIN_F3" )
   END_RUNG
   RUNG wire#w2
      I_Contact( "DB_Status".Up_Called_F3 )
      R_Coil( "Q_BTT_Up_F3" )
   END_RUNG
   RUNG wire#w2
      I_Contact( "DB_Status".Down_Called_F3 )
      R_Coil( "Q_BTT_Down_F3" )
   END_RUNG
   // the same network as SCL:
   IF NOT "AlwaysFALSE" AND "M_BTT_CABINET_F3" THEN "Q_BTT_CABIN_F3" := TRUE; END_IF;
   IF NOT "AlwaysFALSE" AND "M_BTT_UP_F3" THEN "Q_BTT_Up_F3" := TRUE; END_IF;
   IF NOT "AlwaysFALSE" AND "M_BTT_DOWN_F3" THEN "Q_BTT_Down_F3" := TRUE; END_IF;
   #_w1 := NOT "AlwaysFALSE" AND "DB_Status".LS_F3;
   IF #_w1 THEN "Q_BTT_CABIN_F3" := FALSE; END_IF;
   IF #_w1 AND NOT "DB_Status".Up_Called_F3 THEN "Q_BTT_Up_F3" := FALSE; END_IF;
   IF #_w1 AND NOT "DB_Status".Down_Called_F3 THEN "Q_BTT_Down_F3" := FALSE; END_IF;
END_REGION

REGION Network 5: ĐÈN NÚT NHẤN TẦNG 4
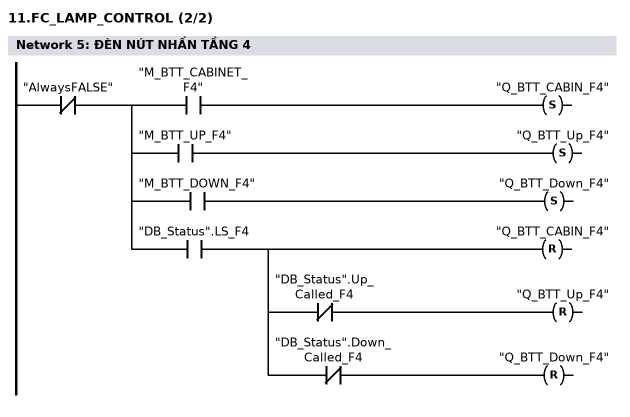
   RUNG wire#powerrail
      I_Contact( "AlwaysFALSE" )
      wire#w1
      Contact( "M_BTT_CABINET_F4" )
      S_Coil( "Q_BTT_CABIN_F4" )
   END_RUNG
   RUNG wire#w1
      Contact( "M_BTT_UP_F4" )
      S_Coil( "Q_BTT_Up_F4" )
   END_RUNG
   RUNG wire#w1
      Contact( "M_BTT_DOWN_F4" )
      S_Coil( "Q_BTT_Down_F4" )
   END_RUNG
   RUNG wire#w1
      Contact( "DB_Status".LS_F4 )
      wire#w2
      R_Coil( "Q_BTT_CABIN_F4" )
   END_RUNG
   RUNG wire#w2
      I_Contact( "DB_Status".Up_Called_F4 )
      R_Coil( "Q_BTT_Up_F4" )
   END_RUNG
   RUNG wire#w2
      I_Contact( "DB_Status".Down_Called_F4 )
      R_Coil( "Q_BTT_Down_F4" )
   END_RUNG
   // the same network as SCL:
   IF NOT "AlwaysFALSE" AND "M_BTT_CABINET_F4" THEN "Q_BTT_CABIN_F4" := TRUE; END_IF;
   IF NOT "AlwaysFALSE" AND "M_BTT_UP_F4" THEN "Q_BTT_Up_F4" := TRUE; END_IF;
   IF NOT "AlwaysFALSE" AND "M_BTT_DOWN_F4" THEN "Q_BTT_Down_F4" := TRUE; END_IF;
   #_w1 := NOT "AlwaysFALSE" AND "DB_Status".LS_F4;
   IF #_w1 THEN "Q_BTT_CABIN_F4" := FALSE; END_IF;
   IF #_w1 AND NOT "DB_Status".Up_Called_F4 THEN "Q_BTT_Up_F4" := FALSE; END_IF;
   IF #_w1 AND NOT "DB_Status".Down_Called_F4 THEN "Q_BTT_Down_F4" := FALSE; END_IF;
END_REGION

REGION Network 6: ĐÈN NÚT NHẤN TẦNG 2
END_REGION
END_FUNCTION

FUNCTION "12.FC_FINAL_FLOOR_CALLED" : Void   // FC12, SCL
{ S7_Optimized_Access := 'TRUE' }
VERSION : 0.1
   VAR_INPUT
      Calling_Up_F2 : Bool;
      Calling_Up_F3 : Bool;
      Calling_Up_F4 : Bool;
      Calling_Down_F1 : Bool;
      Calling_Down_F2 : Bool;
      Calling_Down_F3 : Bool;
      Calling_Down_F4 : Bool;
      Upping_F2 : Bool;
      Upping_F3 : Bool;
      Upping_F4 : Bool;
      Downing_F1 : Bool;
      Downing_F2 : Bool;
      Downing_F3 : Bool;
      Downing_F4 : Bool;
   END_VAR
   VAR_OUTPUT
      F_Stop_Cabin : Bool;   // Lệnh dừng cabin
      F_Open_Door : Bool;   // Lệnh mở cửa
      F_Rq_Remove_PRIORITIZE : Bool;   // Yêu cầu xóa ưu tiên
   END_VAR
   VAR_TEMP
      Temp_Pulse : Bool;   // Bit tạm
      Temp_Pulse2 : Bool;
   END_VAR
BEGIN
   // NẾU CÓ LỆNH GỌI LÊN VÀ THANG MÁY ĐANG ĐI XUỐNG, NẾU TẦNG ĐỐ LÀ TẦNG GỌI LÊN CUỐI CÙNG GỌI LÊN
   // >>> THÌ DỪNG THANG MÁY VÀ MỞ CỬA
   // NGƯỢC LẠI
   // NẾU CÓ LỆNH GỌI XUỐNG VÀ THANG MÁY ĐANG ĐI LÊN, NẾU TẦNG ĐỐ LÀ TẦNG GỌI LÊN CUỐI CÙNG GỌI XUỐNG
   // >>> THÌ DỪNG THANG MÁY VÀ MỞ CỬA
   // 

   // F1_UP
   IF #Calling_Down_F1 = 1
       AND #Downing_F1 = 1
       THEN
           "PULSE".FC12_Pulse_Down_F1 := 1;
       ELSE
           "PULSE".FC12_Pulse_Down_F1 := 0;
           ;
   END_IF;
   // F2_UP
   IF #Calling_Up_F2 = 1
       AND #Downing_F2 = 1 THEN
       IF "PRIORITIZE_1" < 21 AND "PRIORITIZE_1" <> 0
           OR "PRIORITIZE_2" < 21 AND "PRIORITIZE_2" <> 0
           OR "PRIORITIZE_3" < 21 AND "PRIORITIZE_3" <> 0
           OR "PRIORITIZE_4" < 21 AND "PRIORITIZE_4" <> 0
           OR "PRIORITIZE_5" < 21 AND "PRIORITIZE_5" <> 0
           OR "PRIORITIZE_6" < 21 AND "PRIORITIZE_6" <> 0
           OR "PRIORITIZE_7" < 21 AND "PRIORITIZE_7" <> 0
           OR "PRIORITIZE_8" < 21 AND "PRIORITIZE_8" <> 0

       THEN
           "PULSE".FC12_Pulse_Up_F2 := 0;
       ELSE
           "PULSE".FC12_Pulse_Up_F2 := 1;
           ;
       END_IF;
   ELSE
       "PULSE".FC12_Pulse_Up_F2 := 0;
   END_IF;

   // F2_DOWN
   IF #Calling_Down_F2 = 1
       AND #Upping_F2 = 1 THEN
       IF "PRIORITIZE_1" > 20 AND "PRIORITIZE_1" <> 0
           OR "PRIORITIZE_2" > 20 AND "PRIORITIZE_2" <> 0
           OR "PRIORITIZE_3" > 20 AND "PRIORITIZE_3" <> 0
           OR "PRIORITIZE_4" > 20 AND "PRIORITIZE_4" <> 0
           OR "PRIORITIZE_5" > 20 AND "PRIORITIZE_5" <> 0
           OR "PRIORITIZE_6" > 20 AND "PRIORITIZE_6" <> 0
           OR "PRIORITIZE_7" > 20 AND "PRIORITIZE_7" <> 0
           OR "PRIORITIZE_8" > 20 AND "PRIORITIZE_8" <> 0


       THEN
           "PULSE".FC12_Pulse_Down_F2 := 0;
       ELSE
           "PULSE".FC12_Pulse_Down_F2 := 1;
           ;
       END_IF;
   ELSE
       "PULSE".FC12_Pulse_Down_F2 := 0;
   END_IF;

   // F3_UP
   IF #Calling_Up_F3 = 1
       AND #Downing_F3 = 1 THEN
       IF "PRIORITIZE_1" < 31 AND "PRIORITIZE_1" <> 0
           OR "PRIORITIZE_2" < 31 AND "PRIORITIZE_2" <> 0
           OR "PRIORITIZE_3" < 31 AND "PRIORITIZE_3" <> 0
           OR "PRIORITIZE_4" < 31 AND "PRIORITIZE_4" <> 0
           OR "PRIORITIZE_5" < 31 AND "PRIORITIZE_5" <> 0
           OR "PRIORITIZE_6" < 31 AND "PRIORITIZE_6" <> 0
           OR "PRIORITIZE_7" < 31 AND "PRIORITIZE_7" <> 0
           OR "PRIORITIZE_8" < 31 AND "PRIORITIZE_8" <> 0

       THEN
           "PULSE".FC12_Pulse_Up_F3 := 0;
       ELSE
           "PULSE".FC12_Pulse_Up_F3 := 1;
           ;
       END_IF;
   ELSE
       "PULSE".FC12_Pulse_Up_F3 := 0;
   END_IF;

   // F3_DOWN
   IF #Calling_Down_F3 = 1
       AND #Upping_F3 = 1 THEN
       IF "PRIORITIZE_1" > 30 AND "PRIORITIZE_1" <> 0
           OR "PRIORITIZE_2" > 30 AND "PRIORITIZE_2" <> 0
           OR "PRIORITIZE_3" > 30 AND "PRIORITIZE_3" <> 0
           OR "PRIORITIZE_4" > 30 AND "PRIORITIZE_4" <> 0
           OR "PRIORITIZE_5" > 30 AND "PRIORITIZE_5" <> 0
           OR "PRIORITIZE_6" > 30 AND "PRIORITIZE_6" <> 0
           OR "PRIORITIZE_7" > 30 AND "PRIORITIZE_7" <> 0
           OR "PRIORITIZE_8" > 30 AND "PRIORITIZE_8" <> 0
           OR "PRIORITIZE_9" > 30 AND "PRIORITIZE_9" <> 0
           OR "PRIORITIZE_10" > 30 AND "PRIORITIZE_10" <> 0
           OR "PRIORITIZE_11" > 30 AND "PRIORITIZE_11" <> 0
           OR "PRIORITIZE_12" > 30 AND "PRIORITIZE_12" <> 0
       THEN
           "PULSE".FC12_Pulse_Down_F3 := 0;
       ELSE
           "PULSE".FC12_Pulse_Down_F3 := 1;
           ;
       END_IF;
   ELSE
       "PULSE".FC12_Pulse_Down_F3 := 0;
   END_IF;

   // F4_UP
   IF #Calling_Up_F4 = 1
       AND #Downing_F4 = 1 THEN
       IF "PRIORITIZE_1" < 41 AND "PRIORITIZE_1" <> 0
           OR "PRIORITIZE_2" < 41 AND "PRIORITIZE_2" <> 0
           OR "PRIORITIZE_3" < 41 AND "PRIORITIZE_3" <> 0
           OR "PRIORITIZE_4" < 41 AND "PRIORITIZE_4" <> 0
           OR "PRIORITIZE_5" < 41 AND "PRIORITIZE_5" <> 0
           OR "PRIORITIZE_6" < 41 AND "PRIORITIZE_6" <> 0
           OR "PRIORITIZE_7" < 41 AND "PRIORITIZE_7" <> 0
           OR "PRIORITIZE_8" < 41 AND "PRIORITIZE_8" <> 0

       THEN
           "PULSE".FC12_Pulse_Up_F4 := 0;
       ELSE
           "PULSE".FC12_Pulse_Up_F4 := 1;
           ;
       END_IF;
   ELSE
       "PULSE".FC12_Pulse_Up_F4 := 0;
   END_IF;

   // F4_DOWN
   IF #Calling_Down_F4 = 1
       AND #Upping_F4 = 1 THEN
       IF "PRIORITIZE_1" > 40 AND "PRIORITIZE_1" <> 0
           OR "PRIORITIZE_2" > 40 AND "PRIORITIZE_2" <> 0
           OR "PRIORITIZE_3" > 40 AND "PRIORITIZE_3" <> 0
           OR "PRIORITIZE_4" > 40 AND "PRIORITIZE_4" <> 0
           OR "PRIORITIZE_5" > 40 AND "PRIORITIZE_5" <> 0
           OR "PRIORITIZE_6" > 40 AND "PRIORITIZE_6" <> 0
           OR "PRIORITIZE_7" > 40 AND "PRIORITIZE_7" <> 0
           OR "PRIORITIZE_8" > 40 AND "PRIORITIZE_8" <> 0

       THEN
           "PULSE".FC12_Pulse_Down_F4 := 0;
       ELSE
           "PULSE".FC12_Pulse_Down_F4 := 1;
           ;
       END_IF;
   ELSE
       "PULSE".FC12_Pulse_Down_F4 := 0;
   END_IF;




   // move to outpu
   // 
   IF "PULSE".FC12_Pulse_Down_F1 = 1
       OR "PULSE".FC12_Pulse_Down_F2 = 1
       OR "PULSE".FC12_Pulse_Down_F3 = 1
       OR "PULSE".FC12_Pulse_Down_F4 = 1
       OR "PULSE".FC12_Pulse_Down_F5 = 1
       OR "PULSE".FC12_Pulse_Down_F6 = 1
       OR "PULSE".FC12_Pulse_Up_F1 = 1
       OR "PULSE".FC12_Pulse_Up_F2 = 1
       OR "PULSE".FC12_Pulse_Up_F3 = 1
       OR "PULSE".FC12_Pulse_Up_F4 = 1

   THEN
       #Temp_Pulse := 1;
   ELSE
       #Temp_Pulse := 0;
       ;
   END_IF;


   "FC12_DELAY_2S".TP(IN:=#Temp_Pulse,
                      PT:=T#5S,
                      Q=>#Temp_Pulse2);

   #F_Open_Door := #Temp_Pulse2;
   #F_Rq_Remove_PRIORITIZE := #Temp_Pulse2;
   #F_Stop_Cabin := #Temp_Pulse2;
END_FUNCTION

FUNCTION "13_MANUAL_MODE" : Void   // FC13, LAD
{ S7_Optimized_Access := 'TRUE' }
VERSION : 0.1
BEGIN

REGION Network 1: CA BIN ĐI LÊN
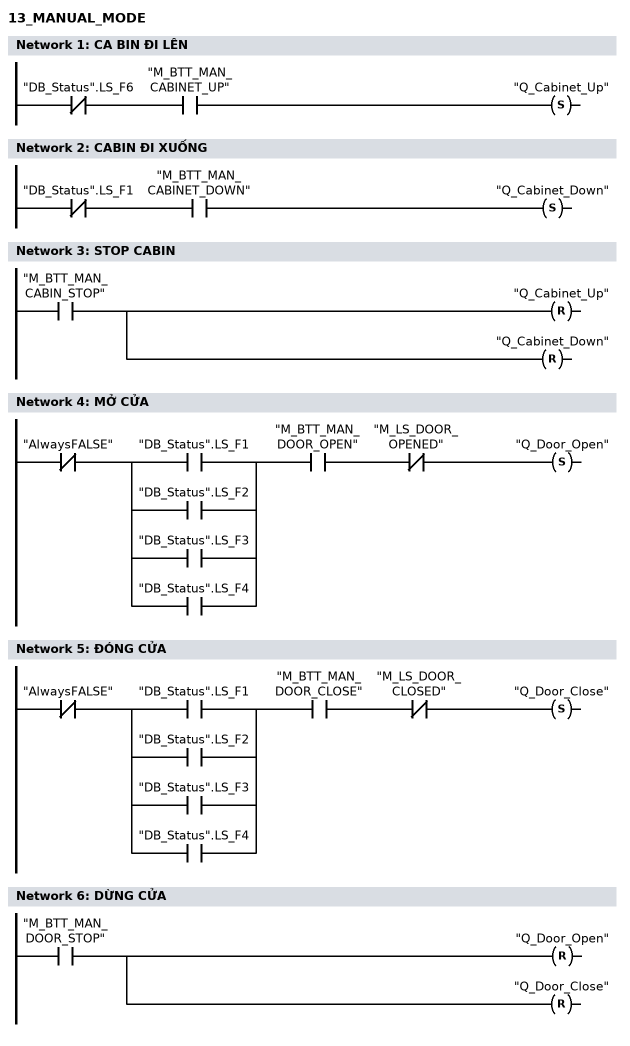
   RUNG wire#powerrail
      I_Contact( "DB_Status".LS_F6 )
      Contact( "M_BTT_MAN_CABINET_UP" )
      S_Coil( "Q_Cabinet_Up" )
   END_RUNG
   // the same network as SCL:
   IF NOT "DB_Status".LS_F6 AND "M_BTT_MAN_CABINET_UP" THEN "Q_Cabinet_Up" := TRUE; END_IF;
END_REGION

REGION Network 2: CABIN ĐI XUỐNG
   RUNG wire#powerrail
      I_Contact( "DB_Status".LS_F1 )
      Contact( "M_BTT_MAN_CABINET_DOWN" )
      S_Coil( "Q_Cabinet_Down" )
   END_RUNG
   // the same network as SCL:
   IF NOT "DB_Status".LS_F1 AND "M_BTT_MAN_CABINET_DOWN" THEN "Q_Cabinet_Down" := TRUE; END_IF;
END_REGION

REGION Network 3: STOP CABIN
   RUNG wire#powerrail
      Contact( "M_BTT_MAN_CABIN_STOP" )
      wire#w1
      R_Coil( "Q_Cabinet_Up" )
   END_RUNG
   RUNG wire#w1
      R_Coil( "Q_Cabinet_Down" )
   END_RUNG
   // the same network as SCL:
   IF "M_BTT_MAN_CABIN_STOP" THEN
       "Q_Cabinet_Up" := FALSE;
       "Q_Cabinet_Down" := FALSE;
   END_IF;
END_REGION

REGION Network 4: MỞ CỬA
   RUNG wire#powerrail
      I_Contact( "AlwaysFALSE" )
      wire#w1
      Contact( "DB_Status".LS_F1 )
      wire#w2
      Contact( "M_BTT_MAN_DOOR_OPEN" )
      I_Contact( "M_LS_DOOR_OPENED" )
      S_Coil( "Q_Door_Open" )
   END_RUNG
   RUNG wire#w1
      Contact( "DB_Status".LS_F2 )
   END_RUNG wire#w2
   RUNG wire#w1
      Contact( "DB_Status".LS_F3 )
   END_RUNG wire#w2
   RUNG wire#w1
      Contact( "DB_Status".LS_F4 )
   END_RUNG wire#w2
   // the same network as SCL:
   IF NOT "AlwaysFALSE" AND ("DB_Status".LS_F1 OR "DB_Status".LS_F2 OR "DB_Status".LS_F3 OR "DB_Status".LS_F4) AND "M_BTT_MAN_DOOR_OPEN" AND NOT "M_LS_DOOR_OPENED" THEN
       "Q_Door_Open" := TRUE;
   END_IF;
END_REGION

REGION Network 5: ĐÓNG CỬA
   RUNG wire#powerrail
      I_Contact( "AlwaysFALSE" )
      wire#w1
      Contact( "DB_Status".LS_F1 )
      wire#w2
      Contact( "M_BTT_MAN_DOOR_CLOSE" )
      I_Contact( "M_LS_DOOR_CLOSED" )
      S_Coil( "Q_Door_Close" )
   END_RUNG
   RUNG wire#w1
      Contact( "DB_Status".LS_F2 )
   END_RUNG wire#w2
   RUNG wire#w1
      Contact( "DB_Status".LS_F3 )
   END_RUNG wire#w2
   RUNG wire#w1
      Contact( "DB_Status".LS_F4 )
   END_RUNG wire#w2
   // the same network as SCL:
   IF NOT "AlwaysFALSE" AND ("DB_Status".LS_F1 OR "DB_Status".LS_F2 OR "DB_Status".LS_F3 OR "DB_Status".LS_F4) AND "M_BTT_MAN_DOOR_CLOSE" AND NOT "M_LS_DOOR_CLOSED" THEN
       "Q_Door_Close" := TRUE;
   END_IF;
END_REGION

REGION Network 6: DỪNG CỬA
   RUNG wire#powerrail
      Contact( "M_BTT_MAN_DOOR_STOP" )
      wire#w1
      R_Coil( "Q_Door_Open" )
   END_RUNG
   RUNG wire#w1
      R_Coil( "Q_Door_Close" )
   END_RUNG
   // the same network as SCL:
   IF "M_BTT_MAN_DOOR_STOP" THEN
       "Q_Door_Open" := FALSE;
       "Q_Door_Close" := FALSE;
   END_IF;
END_REGION
END_FUNCTION

FUNCTION "Block_1" : Void   // FC14, LAD
{ S7_Optimized_Access := 'TRUE' }
VERSION : 0.1
   VAR_INPUT
      "I_UP F1" : Bool;
      "I_UP F2" : Bool;
      "I_UP F3" : Bool;
      I_DOWN_F2 : Bool;
      I_DOWN_F3 : Bool;
      I_DOWN_F4 : Bool;
      F1 : Bool;
      F2 : Bool;
      F3 : Bool;
      F4 : Bool;
      "Đóng cửa" : Bool;
      "Mở cửa" : Bool;
      Ibit_cabinit : Bool;
   END_VAR
BEGIN

REGION Network 1
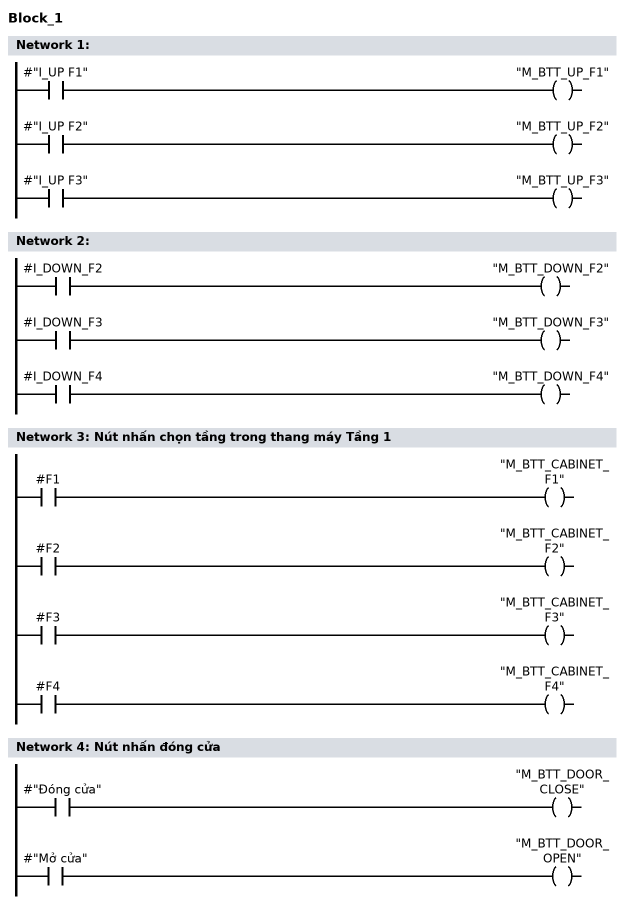
   RUNG wire#powerrail
      Contact( #"I_UP F1" )
      Coil( "M_BTT_UP_F1" )
   END_RUNG
   RUNG wire#powerrail
      Contact( #"I_UP F2" )
      Coil( "M_BTT_UP_F2" )
   END_RUNG
   RUNG wire#powerrail
      Contact( #"I_UP F3" )
      Coil( "M_BTT_UP_F3" )
   END_RUNG
   // the same network as SCL:
   "M_BTT_UP_F1" := #"I_UP F1";
   "M_BTT_UP_F2" := #"I_UP F2";
   "M_BTT_UP_F3" := #"I_UP F3";
END_REGION

REGION Network 2
   RUNG wire#powerrail
      Contact( #I_DOWN_F2 )
      Coil( "M_BTT_DOWN_F2" )
   END_RUNG
   RUNG wire#powerrail
      Contact( #I_DOWN_F3 )
      Coil( "M_BTT_DOWN_F3" )
   END_RUNG
   RUNG wire#powerrail
      Contact( #I_DOWN_F4 )
      Coil( "M_BTT_DOWN_F4" )
   END_RUNG
   // the same network as SCL:
   "M_BTT_DOWN_F2" := #I_DOWN_F2;
   "M_BTT_DOWN_F3" := #I_DOWN_F3;
   "M_BTT_DOWN_F4" := #I_DOWN_F4;
END_REGION

REGION Network 3: Nút nhấn chọn tầng trong thang máy Tầng 1
   RUNG wire#powerrail
      Contact( #F1 )
      Coil( "M_BTT_CABINET_F1" )
   END_RUNG
   RUNG wire#powerrail
      Contact( #F2 )
      Coil( "M_BTT_CABINET_F2" )
   END_RUNG
   RUNG wire#powerrail
      Contact( #F3 )
      Coil( "M_BTT_CABINET_F3" )
   END_RUNG
   RUNG wire#powerrail
      Contact( #F4 )
      Coil( "M_BTT_CABINET_F4" )
   END_RUNG
   // the same network as SCL:
   "M_BTT_CABINET_F1" := #F1;
   "M_BTT_CABINET_F2" := #F2;
   "M_BTT_CABINET_F3" := #F3;
   "M_BTT_CABINET_F4" := #F4;
END_REGION

REGION Network 4: Nút nhấn đóng cửa
   RUNG wire#powerrail
      Contact( #"Đóng cửa" )
      Coil( "M_BTT_DOOR_CLOSE" )
   END_RUNG
   RUNG wire#powerrail
      Contact( #"Mở cửa" )
      Coil( "M_BTT_DOOR_OPEN" )
   END_RUNG
   // the same network as SCL:
   "M_BTT_DOOR_CLOSE" := #"Đóng cửa";
   "M_BTT_DOOR_OPEN" := #"Mở cửa";
END_REGION
END_FUNCTION

ORGANIZATION_BLOCK "Main"   // OB1, LAD, ProgramCycle
TITLE = "Main Program Sweep (Cycle)"
{ S7_Optimized_Access := 'TRUE' }
VERSION : 0.1
   VAR_INPUT
      Initial_Call : Bool;   // Initial call of this OB
      Remanence : Bool;   // =True, if remanent data are available
   END_VAR
   VAR_TEMP   // added for the SCL form of the ladder/FBD networks
      _w1 : Bool;
      _w2 : Bool;
      _w3 : Bool;
      _w4 : Bool;
      _w5 : Bool;
      _w6 : Bool;
      _w7 : Bool;
   END_VAR
BEGIN

REGION Network 1: MOVING INPUT TO M
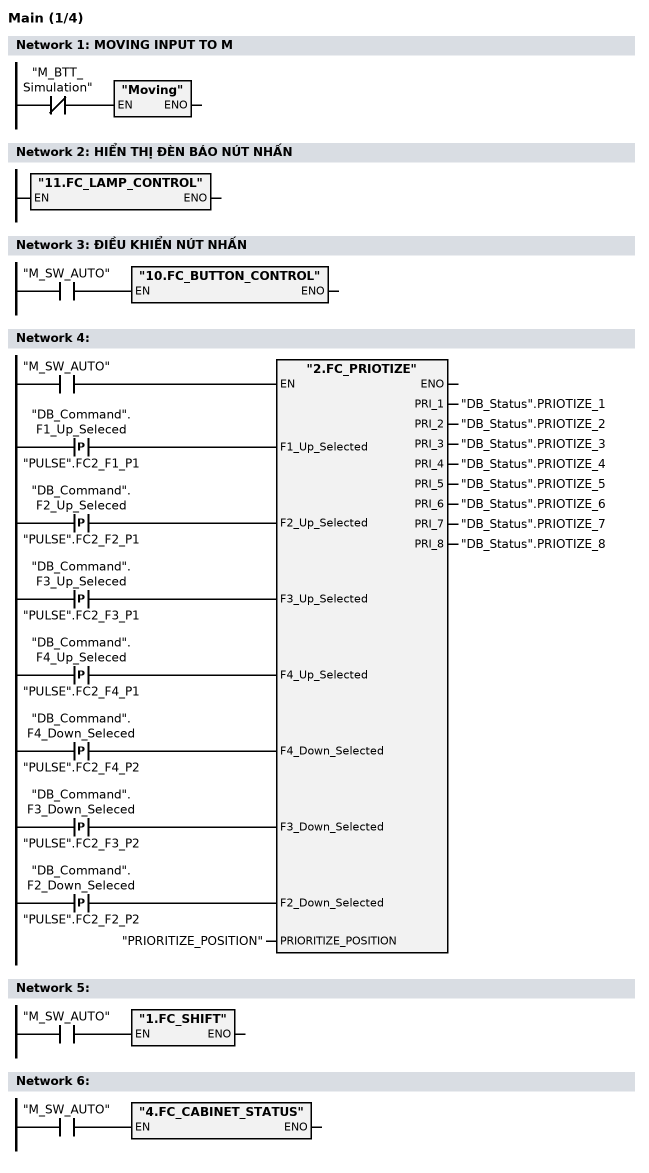
   RUNG wire#powerrail
      I_Contact( "M_BTT_Simulation" )
      "Moving"()
   END_RUNG
   // the same network as SCL:
   IF NOT "M_BTT_Simulation" THEN "Moving"(); END_IF;
END_REGION

REGION Network 2: HIỂN THỊ ĐÈN BÁO NÚT NHẤN
   RUNG wire#powerrail
      "11.FC_LAMP_CONTROL"()
   END_RUNG
   // the same network as SCL:
   "11.FC_LAMP_CONTROL"();
END_REGION

REGION Network 3: ĐIỀU KHIỂN NÚT NHẤN
   RUNG wire#powerrail
      Contact( "M_SW_AUTO" )
      "10.FC_BUTTON_CONTROL"()
   END_RUNG
   // the same network as SCL:
   IF "M_SW_AUTO" THEN "10.FC_BUTTON_CONTROL"(); END_IF;
END_REGION

REGION Network 4
   RUNG wire#powerrail
      Contact( "M_SW_AUTO" )
      "2.FC_PRIOTIZE"(F1_Up_Selected := wire#w1, F2_Up_Selected := wire#w2, F3_Up_Selected := wire#w3, F4_Up_Selected := wire#w4, F4_Down_Selected := wire#w5, F3_Down_Selected := wire#w6, F2_Down_Selected := wire#w7, PRIORITIZE_POSITION := "PRIORITIZE_POSITION", PRI_1 => "DB_Status".PRIOTIZE_1, PRI_2 => "DB_Status".PRIOTIZE_2, PRI_3 => "DB_Status".PRIOTIZE_3, PRI_4 => "DB_Status".PRIOTIZE_4, PRI_5 => "DB_Status".PRIOTIZE_5, PRI_6 => "DB_Status".PRIOTIZE_6, PRI_7 => "DB_Status".PRIOTIZE_7, PRI_8 => "DB_Status".PRIOTIZE_8)
   END_RUNG
   RUNG wire#powerrail
      P_Contact(operand := "DB_Command".F1_Up_Seleced, bit := "PULSE".FC2_F1_P1)
   END_RUNG wire#w1
   RUNG wire#powerrail
      P_Contact(operand := "DB_Command".F2_Up_Seleced, bit := "PULSE".FC2_F2_P1)
   END_RUNG wire#w2
   RUNG wire#powerrail
      P_Contact(operand := "DB_Command".F3_Up_Seleced, bit := "PULSE".FC2_F3_P1)
   END_RUNG wire#w3
   RUNG wire#powerrail
      P_Contact(operand := "DB_Command".F4_Up_Seleced, bit := "PULSE".FC2_F4_P1)
   END_RUNG wire#w4
   RUNG wire#powerrail
      P_Contact(operand := "DB_Command".F4_Down_Seleced, bit := "PULSE".FC2_F4_P2)
   END_RUNG wire#w5
   RUNG wire#powerrail
      P_Contact(operand := "DB_Command".F3_Down_Seleced, bit := "PULSE".FC2_F3_P2)
   END_RUNG wire#w6
   RUNG wire#powerrail
      P_Contact(operand := "DB_Command".F2_Down_Seleced, bit := "PULSE".FC2_F2_P2)
   END_RUNG wire#w7
   // the same network as SCL:
   #_w1 := "DB_Command".F1_Up_Seleced AND NOT "PULSE".FC2_F1_P1;   // rising edge of "DB_Command".F1_Up_Seleced
   "PULSE".FC2_F1_P1 := "DB_Command".F1_Up_Seleced;
   #_w2 := "DB_Command".F2_Up_Seleced AND NOT "PULSE".FC2_F2_P1;   // rising edge of "DB_Command".F2_Up_Seleced
   "PULSE".FC2_F2_P1 := "DB_Command".F2_Up_Seleced;
   #_w3 := "DB_Command".F3_Up_Seleced AND NOT "PULSE".FC2_F3_P1;   // rising edge of "DB_Command".F3_Up_Seleced
   "PULSE".FC2_F3_P1 := "DB_Command".F3_Up_Seleced;
   #_w4 := "DB_Command".F4_Up_Seleced AND NOT "PULSE".FC2_F4_P1;   // rising edge of "DB_Command".F4_Up_Seleced
   "PULSE".FC2_F4_P1 := "DB_Command".F4_Up_Seleced;
   #_w5 := "DB_Command".F4_Down_Seleced AND NOT "PULSE".FC2_F4_P2;   // rising edge of "DB_Command".F4_Down_Seleced
   "PULSE".FC2_F4_P2 := "DB_Command".F4_Down_Seleced;
   #_w6 := "DB_Command".F3_Down_Seleced AND NOT "PULSE".FC2_F3_P2;   // rising edge of "DB_Command".F3_Down_Seleced
   "PULSE".FC2_F3_P2 := "DB_Command".F3_Down_Seleced;
   #_w7 := "DB_Command".F2_Down_Seleced AND NOT "PULSE".FC2_F2_P2;   // rising edge of "DB_Command".F2_Down_Seleced
   "PULSE".FC2_F2_P2 := "DB_Command".F2_Down_Seleced;
   IF "M_SW_AUTO" THEN
       "2.FC_PRIOTIZE"(F1_Up_Selected := #_w1,
                       F2_Up_Selected := #_w2,
                       F3_Up_Selected := #_w3,
                       F4_Up_Selected := #_w4,
                       F4_Down_Selected := #_w5,
                       F3_Down_Selected := #_w6,
                       F2_Down_Selected := #_w7,
                       PRIORITIZE_POSITION := "PRIORITIZE_POSITION",
                       PRI_1 => "DB_Status".PRIOTIZE_1,
                       PRI_2 => "DB_Status".PRIOTIZE_2,
                       PRI_3 => "DB_Status".PRIOTIZE_3,
                       PRI_4 => "DB_Status".PRIOTIZE_4,
                       PRI_5 => "DB_Status".PRIOTIZE_5,
                       PRI_6 => "DB_Status".PRIOTIZE_6,
                       PRI_7 => "DB_Status".PRIOTIZE_7,
                       PRI_8 => "DB_Status".PRIOTIZE_8);
   END_IF;
END_REGION

REGION Network 5
   RUNG wire#powerrail
      Contact( "M_SW_AUTO" )
      "1.FC_SHIFT"()
   END_RUNG
   // the same network as SCL:
   IF "M_SW_AUTO" THEN "1.FC_SHIFT"(); END_IF;
END_REGION

